(* IEC 61131-3 sources: mect_apps/TPAC1007_04_AA/Octopus_Head_PLC, 25 files *)

(* ---- Crosstable.gvl ---- *)
VAR_GLOBAL
PRODUCT_ID AT %QD0.4:UDINT;
SERIAL_NUMBER AT %QD0.8:UDINT;
TEST_ID AT %QW0.12:UINT;
TEST_STEP AT %QW0.16:UINT;
TEST_STEP_MAX AT %QW0.20:UINT;
TEST_DATE AT %QD0.24:UDINT;
TEST_TIME AT %QD0.28:UDINT;
TEST_DURATION AT %QD0.32:UDINT;
AUTOMATIC AT %IX0.772.0:BOOL;
DO_REPEAT AT %IX0.776.0:BOOL;
DO_RELOAD AT %IX0.780.0:BOOL;
STATUS AT %QW0.784:UINT;
RESULT AT %QW0.788:INT;
RESULTS_OK AT %QW0.792:UINT;
RESULTS_NG AT %QW0.796:UINT;
RTU_HeartBeat AT %ID0.832:UDINT;
RTU_DigOut_1 AT %QX0.840.0:BOOL;
RTU_DigOut_2 AT %QX0.844.0:BOOL;
RTU_DigOut_3 AT %QX0.848.0:BOOL;
RTU_DigOut_4 AT %QX0.852.0:BOOL;
RTU_DigOut_5 AT %QX0.856.0:BOOL;
RTU_DigOut_6 AT %QX0.860.0:BOOL;
RTU_DigOut_7 AT %QX0.864.0:BOOL;
RTU_DigOut_8 AT %QX0.868.0:BOOL;
RTU_DigOut_9 AT %QX0.872.0:BOOL;
RTU_DigOut_10 AT %QX0.876.0:BOOL;
RTU_DigOut_11 AT %QX0.880.0:BOOL;
RTU_DigOut_12 AT %QX0.884.0:BOOL;
RTU_DigOut_13 AT %QX0.888.0:BOOL;
RTU_DigOut_14 AT %QX0.892.0:BOOL;
RTU_DigOut_15 AT %QX0.896.0:BOOL;
RTU_DigOut_16 AT %QX0.900.0:BOOL;
RTU_DigIn_1 AT %IX0.908.0:BOOL;
RTU_DigIn_2 AT %IX0.912.0:BOOL;
RTU_DigIn_3 AT %IX0.916.0:BOOL;
RTU_DigIn_4 AT %IX0.920.0:BOOL;
RTU_DigIn_5 AT %IX0.924.0:BOOL;
RTU_DigIn_6 AT %IX0.928.0:BOOL;
RTU_DigIn_7 AT %IX0.932.0:BOOL;
RTU_DigIn_8 AT %IX0.936.0:BOOL;
RTU_DigIn_9 AT %IX0.940.0:BOOL;
RTU_DigIn_10 AT %IX0.944.0:BOOL;
RTU_DigIn_11 AT %IX0.948.0:BOOL;
RTU_DigIn_12 AT %IX0.952.0:BOOL;
RTU_DigIn_13 AT %IX0.956.0:BOOL;
RTU_DigIn_14 AT %IX0.960.0:BOOL;
RTU_DigIn_15 AT %IX0.964.0:BOOL;
RTU_DigIn_16 AT %IX0.968.0:BOOL;
RTU_Tamb AT %IW0.976:INT;
RTU_AnInConf_1 AT %QW0.980:UINT;
RTU_AnInConf_2 AT %QW0.984:UINT;
RTU_AnIn_1 AT %IW0.988:INT;
RTU_AnIn_2 AT %IW0.992:INT;
RTU_LocDigDir_1 AT %QX0.996.0:BOOL;
RTU_LocDigDir_2 AT %QX0.1000.0:BOOL;
RTU_LocDigDir_3 AT %QX0.1004.0:BOOL;
RTU_LocDigDir_4 AT %QX0.1008.0:BOOL;
RTU_LocDigDir_5 AT %QX0.1012.0:BOOL;
RTU_LocDigDir_6 AT %QX0.1016.0:BOOL;
RTU_LocDigDir_7 AT %QX0.1020.0:BOOL;
RTU_LocDigDir_8 AT %QX0.1024.0:BOOL;
RTU_LocDigIn_1 AT %IX0.1028.0:BOOL;
RTU_LocDigIn_2 AT %IX0.1032.0:BOOL;
RTU_LocDigIn_3 AT %IX0.1036.0:BOOL;
RTU_LocDigIn_4 AT %IX0.1040.0:BOOL;
RTU_LocDigIn_5 AT %IX0.1044.0:BOOL;
RTU_LocDigIn_6 AT %IX0.1048.0:BOOL;
RTU_LocDigIn_7 AT %IX0.1052.0:BOOL;
RTU_LocDigIn_8 AT %IX0.1056.0:BOOL;
RTU_LocDigOut_1 AT %QX0.1060.0:BOOL;
RTU_LocDigOut_2 AT %QX0.1064.0:BOOL;
RTU_LocDigOut_3 AT %QX0.1068.0:BOOL;
RTU_LocDigOut_4 AT %QX0.1072.0:BOOL;
RTU_LocDigOut_5 AT %QX0.1076.0:BOOL;
RTU_LocDigOut_6 AT %QX0.1080.0:BOOL;
RTU_LocDigOut_7 AT %QX0.1084.0:BOOL;
RTU_LocDigOut_8 AT %QX0.1088.0:BOOL;
TST_DigIn_1 AT %QX0.4004.0:BOOL;
TST_DigIn_2 AT %QX0.4008.0:BOOL;
TST_DigIn_3 AT %QX0.4012.0:BOOL;
TST_DigIn_4 AT %QX0.4016.0:BOOL;
TST_DigIn_5 AT %QX0.4020.0:BOOL;
TST_DigIn_6 AT %QX0.4024.0:BOOL;
TST_DigIn_7 AT %QX0.4028.0:BOOL;
TST_DigIn_8 AT %QX0.4032.0:BOOL;
TST_DigIn_9 AT %QX0.4036.0:BOOL;
TST_DigIn_10 AT %QX0.4040.0:BOOL;
TST_DigIn_11 AT %QX0.4044.0:BOOL;
TST_DigIn_12 AT %QX0.4048.0:BOOL;
TST_DigIn_13 AT %QX0.4052.0:BOOL;
TST_DigIn_14 AT %QX0.4056.0:BOOL;
TST_DigIn_15 AT %QX0.4060.0:BOOL;
TST_DigIn_16 AT %QX0.4064.0:BOOL;
VAL_DigIn_1 AT %QX0.4068.0:BOOL;
VAL_DigIn_2 AT %QX0.4072.0:BOOL;
VAL_DigIn_3 AT %QX0.4076.0:BOOL;
VAL_DigIn_4 AT %QX0.4080.0:BOOL;
VAL_DigIn_5 AT %QX0.4084.0:BOOL;
VAL_DigIn_6 AT %QX0.4088.0:BOOL;
VAL_DigIn_7 AT %QX0.4092.0:BOOL;
VAL_DigIn_8 AT %QX0.4096.0:BOOL;
VAL_DigIn_9 AT %QX0.4100.0:BOOL;
VAL_DigIn_10 AT %QX0.4104.0:BOOL;
VAL_DigIn_11 AT %QX0.4108.0:BOOL;
VAL_DigIn_12 AT %QX0.4112.0:BOOL;
VAL_DigIn_13 AT %QX0.4116.0:BOOL;
VAL_DigIn_14 AT %QX0.4120.0:BOOL;
VAL_DigIn_15 AT %QX0.4124.0:BOOL;
VAL_DigIn_16 AT %QX0.4128.0:BOOL;
RES_DigIn_1 AT %QX0.4132.0:BOOL;
RES_DigIn_2 AT %QX0.4136.0:BOOL;
RES_DigIn_3 AT %QX0.4140.0:BOOL;
RES_DigIn_4 AT %QX0.4144.0:BOOL;
RES_DigIn_5 AT %QX0.4148.0:BOOL;
RES_DigIn_6 AT %QX0.4152.0:BOOL;
RES_DigIn_7 AT %QX0.4156.0:BOOL;
RES_DigIn_8 AT %QX0.4160.0:BOOL;
RES_DigIn_9 AT %QX0.4164.0:BOOL;
RES_DigIn_10 AT %QX0.4168.0:BOOL;
RES_DigIn_11 AT %QX0.4172.0:BOOL;
RES_DigIn_12 AT %QX0.4176.0:BOOL;
RES_DigIn_13 AT %QX0.4180.0:BOOL;
RES_DigIn_14 AT %QX0.4184.0:BOOL;
RES_DigIn_15 AT %QX0.4188.0:BOOL;
RES_DigIn_16 AT %QX0.4192.0:BOOL;
OK_DigIn_1 AT %QX0.4196.0:BOOL;
OK_DigIn_2 AT %QX0.4200.0:BOOL;
OK_DigIn_3 AT %QX0.4204.0:BOOL;
OK_DigIn_4 AT %QX0.4208.0:BOOL;
OK_DigIn_5 AT %QX0.4212.0:BOOL;
OK_DigIn_6 AT %QX0.4216.0:BOOL;
OK_DigIn_7 AT %QX0.4220.0:BOOL;
OK_DigIn_8 AT %QX0.4224.0:BOOL;
OK_DigIn_9 AT %QX0.4228.0:BOOL;
OK_DigIn_10 AT %QX0.4232.0:BOOL;
OK_DigIn_11 AT %QX0.4236.0:BOOL;
OK_DigIn_12 AT %QX0.4240.0:BOOL;
OK_DigIn_13 AT %QX0.4244.0:BOOL;
OK_DigIn_14 AT %QX0.4248.0:BOOL;
OK_DigIn_15 AT %QX0.4252.0:BOOL;
OK_DigIn_16 AT %QX0.4256.0:BOOL;
TST_DigOut_1 AT %QX0.4260.0:BOOL;
TST_DigOut_2 AT %QX0.4264.0:BOOL;
TST_DigOut_3 AT %QX0.4268.0:BOOL;
TST_DigOut_4 AT %QX0.4272.0:BOOL;
TST_DigOut_5 AT %QX0.4276.0:BOOL;
TST_DigOut_6 AT %QX0.4280.0:BOOL;
TST_DigOut_7 AT %QX0.4284.0:BOOL;
TST_DigOut_8 AT %QX0.4288.0:BOOL;
TST_DigOut_9 AT %QX0.4292.0:BOOL;
TST_DigOut_10 AT %QX0.4296.0:BOOL;
TST_DigOut_11 AT %QX0.4300.0:BOOL;
TST_DigOut_12 AT %QX0.4304.0:BOOL;
TST_DigOut_13 AT %QX0.4308.0:BOOL;
TST_DigOut_14 AT %QX0.4312.0:BOOL;
TST_DigOut_15 AT %QX0.4316.0:BOOL;
TST_DigOut_16 AT %QX0.4320.0:BOOL;
VAL_DigOut_1 AT %QX0.4324.0:BOOL;
VAL_DigOut_2 AT %QX0.4328.0:BOOL;
VAL_DigOut_3 AT %QX0.4332.0:BOOL;
VAL_DigOut_4 AT %QX0.4336.0:BOOL;
VAL_DigOut_5 AT %QX0.4340.0:BOOL;
VAL_DigOut_6 AT %QX0.4344.0:BOOL;
VAL_DigOut_7 AT %QX0.4348.0:BOOL;
VAL_DigOut_8 AT %QX0.4352.0:BOOL;
VAL_DigOut_9 AT %QX0.4356.0:BOOL;
VAL_DigOut_10 AT %QX0.4360.0:BOOL;
VAL_DigOut_11 AT %QX0.4364.0:BOOL;
VAL_DigOut_12 AT %QX0.4368.0:BOOL;
VAL_DigOut_13 AT %QX0.4372.0:BOOL;
VAL_DigOut_14 AT %QX0.4376.0:BOOL;
VAL_DigOut_15 AT %QX0.4380.0:BOOL;
VAL_DigOut_16 AT %QX0.4384.0:BOOL;
RES_DigOut_1 AT %QX0.4388.0:BOOL;
RES_DigOut_2 AT %QX0.4392.0:BOOL;
RES_DigOut_3 AT %QX0.4396.0:BOOL;
RES_DigOut_4 AT %QX0.4400.0:BOOL;
RES_DigOut_5 AT %QX0.4404.0:BOOL;
RES_DigOut_6 AT %QX0.4408.0:BOOL;
RES_DigOut_7 AT %QX0.4412.0:BOOL;
RES_DigOut_8 AT %QX0.4416.0:BOOL;
RES_DigOut_9 AT %QX0.4420.0:BOOL;
RES_DigOut_10 AT %QX0.4424.0:BOOL;
RES_DigOut_11 AT %QX0.4428.0:BOOL;
RES_DigOut_12 AT %QX0.4432.0:BOOL;
RES_DigOut_13 AT %QX0.4436.0:BOOL;
RES_DigOut_14 AT %QX0.4440.0:BOOL;
RES_DigOut_15 AT %QX0.4444.0:BOOL;
RES_DigOut_16 AT %QX0.4448.0:BOOL;
OK_DigOut_1 AT %QX0.4452.0:BOOL;
OK_DigOut_2 AT %QX0.4456.0:BOOL;
OK_DigOut_3 AT %QX0.4460.0:BOOL;
OK_DigOut_4 AT %QX0.4464.0:BOOL;
OK_DigOut_5 AT %QX0.4468.0:BOOL;
OK_DigOut_6 AT %QX0.4472.0:BOOL;
OK_DigOut_7 AT %QX0.4476.0:BOOL;
OK_DigOut_8 AT %QX0.4480.0:BOOL;
OK_DigOut_9 AT %QX0.4484.0:BOOL;
OK_DigOut_10 AT %QX0.4488.0:BOOL;
OK_DigOut_11 AT %QX0.4492.0:BOOL;
OK_DigOut_12 AT %QX0.4496.0:BOOL;
OK_DigOut_13 AT %QX0.4500.0:BOOL;
OK_DigOut_14 AT %QX0.4504.0:BOOL;
OK_DigOut_15 AT %QX0.4508.0:BOOL;
OK_DigOut_16 AT %QX0.4512.0:BOOL;
TST_AnIn_1 AT %QX0.4516.0:BOOL;
TST_AnIn_2 AT %QX0.4520.0:BOOL;
TST_AnIn_3 AT %QX0.4524.0:BOOL;
TST_AnIn_4 AT %QX0.4528.0:BOOL;
TST_AnIn_5 AT %QX0.4532.0:BOOL;
TST_AnIn_6 AT %QX0.4536.0:BOOL;
TST_AnIn_7 AT %QX0.4540.0:BOOL;
TST_AnIn_8 AT %QX0.4544.0:BOOL;
TST_AnIn_9 AT %QX0.4548.0:BOOL;
TST_AnIn_10 AT %QX0.4552.0:BOOL;
TST_AnIn_11 AT %QX0.4556.0:BOOL;
TST_AnIn_12 AT %QX0.4560.0:BOOL;
VAL_AnIn_1 AT %QW0.4564:INT;
VAL_AnIn_2 AT %QW0.4568:INT;
VAL_AnIn_3 AT %QW0.4572:INT;
VAL_AnIn_4 AT %QW0.4576:INT;
VAL_AnIn_5 AT %QW0.4580:INT;
VAL_AnIn_6 AT %QW0.4584:INT;
VAL_AnIn_7 AT %QW0.4588:INT;
VAL_AnIn_8 AT %QW0.4592:INT;
VAL_AnIn_9 AT %QW0.4596:INT;
VAL_AnIn_10 AT %QW0.4600:INT;
VAL_AnIn_11 AT %QW0.4604:INT;
VAL_AnIn_12 AT %QW0.4608:INT;
VAL_AnInConf_1 AT %QW0.4612:UINT;
VAL_AnInConf_2 AT %QW0.4616:UINT;
VAL_AnInConf_3 AT %QW0.4620:UINT;
VAL_AnInConf_4 AT %QW0.4624:UINT;
VAL_AnInConf_5 AT %QW0.4628:UINT;
VAL_AnInConf_6 AT %QW0.4632:UINT;
VAL_AnInConf_7 AT %QW0.4636:UINT;
VAL_AnInConf_8 AT %QW0.4640:UINT;
VAL_AnInConf_9 AT %QW0.4644:UINT;
VAL_AnInConf_10 AT %QW0.4648:UINT;
VAL_AnInConf_11 AT %QW0.4652:UINT;
VAL_AnInConf_12 AT %QW0.4656:UINT;
VAL_AnInFltr_1 AT %QW0.4660:UINT;
VAL_AnInFltr_2 AT %QW0.4664:UINT;
VAL_AnInFltr_3 AT %QW0.4668:UINT;
VAL_AnInFltr_4 AT %QW0.4672:UINT;
VAL_AnInFltr_5 AT %QW0.4676:UINT;
VAL_AnInFltr_6 AT %QW0.4680:UINT;
VAL_AnInFltr_7 AT %QW0.4684:UINT;
VAL_AnInFltr_8 AT %QW0.4688:UINT;
VAL_AnInFltr_9 AT %QW0.4692:UINT;
VAL_AnInFltr_10 AT %QW0.4696:UINT;
VAL_AnInFltr_11 AT %QW0.4700:UINT;
VAL_AnInFltr_12 AT %QW0.4704:UINT;
RES_AnIn_1 AT %QW0.4708:INT;
RES_AnIn_2 AT %QW0.4712:INT;
RES_AnIn_3 AT %QW0.4716:INT;
RES_AnIn_4 AT %QW0.4720:INT;
RES_AnIn_5 AT %QW0.4724:INT;
RES_AnIn_6 AT %QW0.4728:INT;
RES_AnIn_7 AT %QW0.4732:INT;
RES_AnIn_8 AT %QW0.4736:INT;
RES_AnIn_9 AT %QW0.4740:INT;
RES_AnIn_10 AT %QW0.4744:INT;
RES_AnIn_11 AT %QW0.4748:INT;
RES_AnIn_12 AT %QW0.4752:INT;
RES_AnInStts_1 AT %QW0.4756:INT;
RES_AnInStts_2 AT %QW0.4760:INT;
RES_AnInStts_3 AT %QW0.4764:INT;
RES_AnInStts_4 AT %QW0.4768:INT;
RES_AnInStts_5 AT %QW0.4772:INT;
RES_AnInStts_6 AT %QW0.4776:INT;
RES_AnInStts_7 AT %QW0.4780:INT;
RES_AnInStts_8 AT %QW0.4784:INT;
RES_AnInStts_9 AT %QW0.4788:INT;
RES_AnInStts_10 AT %QW0.4792:INT;
RES_AnInStts_11 AT %QW0.4796:INT;
RES_AnInStts_12 AT %QW0.4800:INT;
OK_AnIn_1 AT %QX0.4804.0:BOOL;
OK_AnIn_2 AT %QX0.4808.0:BOOL;
OK_AnIn_3 AT %QX0.4812.0:BOOL;
OK_AnIn_4 AT %QX0.4816.0:BOOL;
OK_AnIn_5 AT %QX0.4820.0:BOOL;
OK_AnIn_6 AT %QX0.4824.0:BOOL;
OK_AnIn_7 AT %QX0.4828.0:BOOL;
OK_AnIn_8 AT %QX0.4832.0:BOOL;
OK_AnIn_9 AT %QX0.4836.0:BOOL;
OK_AnIn_10 AT %QX0.4840.0:BOOL;
OK_AnIn_11 AT %QX0.4844.0:BOOL;
OK_AnIn_12 AT %QX0.4848.0:BOOL;
TST_AnOut_1 AT %QX0.4852.0:BOOL;
TST_AnOut_2 AT %QX0.4856.0:BOOL;
TST_AnOut_3 AT %QX0.4860.0:BOOL;
TST_AnOut_4 AT %QX0.4864.0:BOOL;
VAL_AnOut_1 AT %QW0.4868:INT;
VAL_AnOut_2 AT %QW0.4872:INT;
VAL_AnOut_3 AT %QW0.4876:INT;
VAL_AnOut_4 AT %QW0.4880:INT;
VAL_AnOutConf_1 AT %QW0.4884:UINT;
VAL_AnOutConf_2 AT %QW0.4888:UINT;
VAL_AnOutConf_3 AT %QW0.4892:UINT;
VAL_AnOutConf_4 AT %QW0.4896:UINT;
RES_AnOut_1 AT %QW0.4900:INT;
RES_AnOut_2 AT %QW0.4904:INT;
RES_AnOut_3 AT %QW0.4908:INT;
RES_AnOut_4 AT %QW0.4912:INT;
RES_AnOutStts_1 AT %QW0.4916:INT;
RES_AnOutStts_2 AT %QW0.4920:INT;
RES_AnOutStts_3 AT %QW0.4924:INT;
RES_AnOutStts_4 AT %QW0.4928:INT;
OK_AnOut_1 AT %QX0.4932.0:BOOL;
OK_AnOut_2 AT %QX0.4936.0:BOOL;
OK_AnOut_3 AT %QX0.4940.0:BOOL;
OK_AnOut_4 AT %QX0.4944.0:BOOL;
TST_Tamb AT %QX0.4948.0:BOOL;
TST_RPM AT %QX0.4952.0:BOOL;
TST_VCC_set AT %QX0.4956.0:BOOL;
TST_mA_max AT %QX0.4960.0:BOOL;
TST_VCC_fbk AT %QX0.4964.0:BOOL;
TST_mA_fbk AT %QX0.4968.0:BOOL;
TST_FWrevision AT %QX0.4972.0:BOOL;
TST_HWconfig AT %QX0.4976.0:BOOL;
VAL_Tamb AT %QW0.4980:INT;
VAL_RPM AT %QW0.4984:UINT;
VAL_VCC_set AT %QW0.4988:INT;
VAL_mA_max AT %QW0.4992:INT;
VAL_VCC_fbk AT %QW0.4996:INT;
VAL_mA_fbk AT %QW0.5000:INT;
VAL_FWrevision AT %QW0.5004:UINT;
VAL_HWconfig AT %QW0.5008:UINT;
RES_Tamb AT %QW0.5012:INT;
RES_RPM AT %QW0.5016:UINT;
RES_VCC_set AT %QW0.5020:INT;
RES_mA_max AT %QW0.5024:INT;
RES_VCC_fbk AT %QW0.5028:INT;
RES_mA_fbk AT %QW0.5032:INT;
RES_FWrevision AT %QW0.5036:UINT;
RES_HWconfig AT %QW0.5040:UINT;
OK_Tamb AT %QX0.5044.0:BOOL;
OK_RPM AT %QX0.5048.0:BOOL;
OK_VCC_set AT %QX0.5052.0:BOOL;
OK_mA_max AT %QX0.5056.0:BOOL;
OK_VCC_fbk AT %QX0.5060.0:BOOL;
OK_mA_fbk AT %QX0.5064.0:BOOL;
OK_FWrevision AT %QX0.5068.0:BOOL;
OK_HWconfig AT %QX0.5072.0:BOOL;
TST_RTUS_WR AT %QX0.5076.0:BOOL;
TST_RTUS_RD AT %QX0.5080.0:BOOL;
TST_RTU1_WR AT %QX0.5084.0:BOOL;
TST_RTU1_RD AT %QX0.5088.0:BOOL;
TST_RTU3_WR AT %QX0.5092.0:BOOL;
TST_RTU3_RD AT %QX0.5096.0:BOOL;
TST_CAN1_WR AT %QX0.5100.0:BOOL;
TST_CAN1_RD AT %QX0.5104.0:BOOL;
VAL_RTUS_WR AT %QX0.5108.0:BOOL;
VAL_RTUS_RD AT %QX0.5112.0:BOOL;
VAL_RTU1_WR AT %QX0.5116.0:BOOL;
VAL_RTU1_RD AT %QX0.5120.0:BOOL;
VAL_RTU3_WR AT %QX0.5124.0:BOOL;
VAL_RTU3_RD AT %QX0.5128.0:BOOL;
VAL_CAN1_WR AT %QX0.5132.0:BOOL;
VAL_CAN1_RD AT %QX0.5136.0:BOOL;
RES_RTUS_WR AT %QX0.5140.0:BOOL;
RES_RTUS_RD AT %QX0.5144.0:BOOL;
RES_RTU1_WR AT %QX0.5148.0:BOOL;
RES_RTU1_RD AT %QX0.5152.0:BOOL;
RES_RTU3_WR AT %QX0.5156.0:BOOL;
RES_RTU3_RD AT %QX0.5160.0:BOOL;
RES_CAN1_WR AT %QX0.5164.0:BOOL;
RES_CAN1_RD AT %QX0.5168.0:BOOL;
OK_RTUS_WR AT %QX0.5172.0:BOOL;
OK_RTUS_RD AT %QX0.5176.0:BOOL;
OK_RTU1_WR AT %QX0.5180.0:BOOL;
OK_RTU1_RD AT %QX0.5184.0:BOOL;
OK_RTU3_WR AT %QX0.5188.0:BOOL;
OK_RTU3_RD AT %QX0.5192.0:BOOL;
OK_CAN1_WR AT %QX0.5196.0:BOOL;
OK_CAN1_RD AT %QX0.5200.0:BOOL;
TEST2_COMMAND AT %QW0.12000:UINT;
TST2_DigIn_1 AT %QX0.12004.0:BOOL;
TST2_DigIn_2 AT %QX0.12008.0:BOOL;
TST2_DigIn_3 AT %QX0.12012.0:BOOL;
TST2_DigIn_4 AT %QX0.12016.0:BOOL;
TST2_DigIn_5 AT %QX0.12020.0:BOOL;
TST2_DigIn_6 AT %QX0.12024.0:BOOL;
TST2_DigIn_7 AT %QX0.12028.0:BOOL;
TST2_DigIn_8 AT %QX0.12032.0:BOOL;
TST2_DigIn_9 AT %QX0.12036.0:BOOL;
TST2_DigIn_10 AT %QX0.12040.0:BOOL;
TST2_DigIn_11 AT %QX0.12044.0:BOOL;
TST2_DigIn_12 AT %QX0.12048.0:BOOL;
TST2_DigIn_13 AT %QX0.12052.0:BOOL;
TST2_DigIn_14 AT %QX0.12056.0:BOOL;
TST2_DigIn_15 AT %QX0.12060.0:BOOL;
TST2_DigIn_16 AT %QX0.12064.0:BOOL;
VAL2_DigIn_1 AT %QX0.12068.0:BOOL;
VAL2_DigIn_2 AT %QX0.12072.0:BOOL;
VAL2_DigIn_3 AT %QX0.12076.0:BOOL;
VAL2_DigIn_4 AT %QX0.12080.0:BOOL;
VAL2_DigIn_5 AT %QX0.12084.0:BOOL;
VAL2_DigIn_6 AT %QX0.12088.0:BOOL;
VAL2_DigIn_7 AT %QX0.12092.0:BOOL;
VAL2_DigIn_8 AT %QX0.12096.0:BOOL;
VAL2_DigIn_9 AT %QX0.12100.0:BOOL;
VAL2_DigIn_10 AT %QX0.12104.0:BOOL;
VAL2_DigIn_11 AT %QX0.12108.0:BOOL;
VAL2_DigIn_12 AT %QX0.12112.0:BOOL;
VAL2_DigIn_13 AT %QX0.12116.0:BOOL;
VAL2_DigIn_14 AT %QX0.12120.0:BOOL;
VAL2_DigIn_15 AT %QX0.12124.0:BOOL;
VAL2_DigIn_16 AT %QX0.12128.0:BOOL;
RES2_DigIn_1 AT %IX0.12132.0:BOOL;
RES2_DigIn_2 AT %IX0.12136.0:BOOL;
RES2_DigIn_3 AT %IX0.12140.0:BOOL;
RES2_DigIn_4 AT %IX0.12144.0:BOOL;
RES2_DigIn_5 AT %IX0.12148.0:BOOL;
RES2_DigIn_6 AT %IX0.12152.0:BOOL;
RES2_DigIn_7 AT %IX0.12156.0:BOOL;
RES2_DigIn_8 AT %IX0.12160.0:BOOL;
RES2_DigIn_9 AT %IX0.12164.0:BOOL;
RES2_DigIn_10 AT %IX0.12168.0:BOOL;
RES2_DigIn_11 AT %IX0.12172.0:BOOL;
RES2_DigIn_12 AT %IX0.12176.0:BOOL;
RES2_DigIn_13 AT %IX0.12180.0:BOOL;
RES2_DigIn_14 AT %IX0.12184.0:BOOL;
RES2_DigIn_15 AT %IX0.12188.0:BOOL;
RES2_DigIn_16 AT %IX0.12192.0:BOOL;
TST2_DigOut_1 AT %QX0.12196.0:BOOL;
TST2_DigOut_2 AT %QX0.12200.0:BOOL;
TST2_DigOut_3 AT %QX0.12204.0:BOOL;
TST2_DigOut_4 AT %QX0.12208.0:BOOL;
TST2_DigOut_5 AT %QX0.12212.0:BOOL;
TST2_DigOut_6 AT %QX0.12216.0:BOOL;
TST2_DigOut_7 AT %QX0.12220.0:BOOL;
TST2_DigOut_8 AT %QX0.12224.0:BOOL;
TST2_DigOut_9 AT %QX0.12228.0:BOOL;
TST2_DigOut_10 AT %QX0.12232.0:BOOL;
TST2_DigOut_11 AT %QX0.12236.0:BOOL;
TST2_DigOut_12 AT %QX0.12240.0:BOOL;
TST2_DigOut_13 AT %QX0.12244.0:BOOL;
TST2_DigOut_14 AT %QX0.12248.0:BOOL;
TST2_DigOut_15 AT %QX0.12252.0:BOOL;
TST2_DigOut_16 AT %QX0.12256.0:BOOL;
VAL2_DigOut_1 AT %QX0.12260.0:BOOL;
VAL2_DigOut_2 AT %QX0.12264.0:BOOL;
VAL2_DigOut_3 AT %QX0.12268.0:BOOL;
VAL2_DigOut_4 AT %QX0.12272.0:BOOL;
VAL2_DigOut_5 AT %QX0.12276.0:BOOL;
VAL2_DigOut_6 AT %QX0.12280.0:BOOL;
VAL2_DigOut_7 AT %QX0.12284.0:BOOL;
VAL2_DigOut_8 AT %QX0.12288.0:BOOL;
VAL2_DigOut_9 AT %QX0.12292.0:BOOL;
VAL2_DigOut_10 AT %QX0.12296.0:BOOL;
VAL2_DigOut_11 AT %QX0.12300.0:BOOL;
VAL2_DigOut_12 AT %QX0.12304.0:BOOL;
VAL2_DigOut_13 AT %QX0.12308.0:BOOL;
VAL2_DigOut_14 AT %QX0.12312.0:BOOL;
VAL2_DigOut_15 AT %QX0.12316.0:BOOL;
VAL2_DigOut_16 AT %QX0.12320.0:BOOL;
TST2_AnIn_1 AT %QX0.12324.0:BOOL;
TST2_AnIn_2 AT %QX0.12328.0:BOOL;
TST2_AnIn_3 AT %QX0.12332.0:BOOL;
TST2_AnIn_4 AT %QX0.12336.0:BOOL;
TST2_AnIn_5 AT %QX0.12340.0:BOOL;
TST2_AnIn_6 AT %QX0.12344.0:BOOL;
TST2_AnIn_7 AT %QX0.12348.0:BOOL;
TST2_AnIn_8 AT %QX0.12352.0:BOOL;
TST2_AnIn_9 AT %QX0.12356.0:BOOL;
TST2_AnIn_10 AT %QX0.12360.0:BOOL;
TST2_AnIn_11 AT %QX0.12364.0:BOOL;
TST2_AnIn_12 AT %QX0.12368.0:BOOL;
VAL2_AnIn_1 AT %QW0.12372:INT;
VAL2_AnIn_2 AT %QW0.12376:INT;
VAL2_AnIn_3 AT %QW0.12380:INT;
VAL2_AnIn_4 AT %QW0.12384:INT;
VAL2_AnIn_5 AT %QW0.12388:INT;
VAL2_AnIn_6 AT %QW0.12392:INT;
VAL2_AnIn_7 AT %QW0.12396:INT;
VAL2_AnIn_8 AT %QW0.12400:INT;
VAL2_AnIn_9 AT %QW0.12404:INT;
VAL2_AnIn_10 AT %QW0.12408:INT;
VAL2_AnIn_11 AT %QW0.12412:INT;
VAL2_AnIn_12 AT %QW0.12416:INT;
VAL2_AnInConf_1 AT %QW0.12420:UINT;
VAL2_AnInConf_2 AT %QW0.12424:UINT;
VAL2_AnInConf_3 AT %QW0.12428:UINT;
VAL2_AnInConf_4 AT %QW0.12432:UINT;
VAL2_AnInConf_5 AT %QW0.12436:UINT;
VAL2_AnInConf_6 AT %QW0.12440:UINT;
VAL2_AnInConf_7 AT %QW0.12444:UINT;
VAL2_AnInConf_8 AT %QW0.12448:UINT;
VAL2_AnInConf_9 AT %QW0.12452:UINT;
VAL2_AnInConf_10 AT %QW0.12456:UINT;
VAL2_AnInConf_11 AT %QW0.12460:UINT;
VAL2_AnInConf_12 AT %QW0.12464:UINT;
VAL2_AnInFltr_1 AT %QW0.12468:UINT;
VAL2_AnInFltr_2 AT %QW0.12472:UINT;
VAL2_AnInFltr_3 AT %QW0.12476:UINT;
VAL2_AnInFltr_4 AT %QW0.12480:UINT;
VAL2_AnInFltr_5 AT %QW0.12484:UINT;
VAL2_AnInFltr_6 AT %QW0.12488:UINT;
VAL2_AnInFltr_7 AT %QW0.12492:UINT;
VAL2_AnInFltr_8 AT %QW0.12496:UINT;
VAL2_AnInFltr_9 AT %QW0.12500:UINT;
VAL2_AnInFltr_10 AT %QW0.12504:UINT;
VAL2_AnInFltr_11 AT %QW0.12508:UINT;
VAL2_AnInFltr_12 AT %QW0.12512:UINT;
RES2_AnIn_1 AT %IW0.12516:INT;
RES2_AnIn_2 AT %IW0.12520:INT;
RES2_AnIn_3 AT %IW0.12524:INT;
RES2_AnIn_4 AT %IW0.12528:INT;
RES2_AnIn_5 AT %IW0.12532:INT;
RES2_AnIn_6 AT %IW0.12536:INT;
RES2_AnIn_7 AT %IW0.12540:INT;
RES2_AnIn_8 AT %IW0.12544:INT;
RES2_AnIn_9 AT %IW0.12548:INT;
RES2_AnIn_10 AT %IW0.12552:INT;
RES2_AnIn_11 AT %IW0.12556:INT;
RES2_AnIn_12 AT %IW0.12560:INT;
RES2_AnInStts_1 AT %IW0.12564:INT;
RES2_AnInStts_2 AT %IW0.12568:INT;
RES2_AnInStts_3 AT %IW0.12572:INT;
RES2_AnInStts_4 AT %IW0.12576:INT;
RES2_AnInStts_5 AT %IW0.12580:INT;
RES2_AnInStts_6 AT %IW0.12584:INT;
RES2_AnInStts_7 AT %IW0.12588:INT;
RES2_AnInStts_8 AT %IW0.12592:INT;
RES2_AnInStts_9 AT %IW0.12596:INT;
RES2_AnInStts_10 AT %IW0.12600:INT;
RES2_AnInStts_11 AT %IW0.12604:INT;
RES2_AnInStts_12 AT %IW0.12608:INT;
TST2_AnOut_1 AT %QX0.12612.0:BOOL;
TST2_AnOut_2 AT %QX0.12616.0:BOOL;
TST2_AnOut_3 AT %QX0.12620.0:BOOL;
TST2_AnOut_4 AT %QX0.12624.0:BOOL;
VAL2_AnOut_1 AT %QW0.12628:INT;
VAL2_AnOut_2 AT %QW0.12632:INT;
VAL2_AnOut_3 AT %QW0.12636:INT;
VAL2_AnOut_4 AT %QW0.12640:INT;
VAL2_AnOutConf_1 AT %QW0.12644:UINT;
VAL2_AnOutConf_2 AT %QW0.12648:UINT;
VAL2_AnOutConf_3 AT %QW0.12652:UINT;
VAL2_AnOutConf_4 AT %QW0.12656:UINT;
RES2_AnOutStts_1 AT %IW0.12660:INT;
RES2_AnOutStts_2 AT %IW0.12664:INT;
RES2_AnOutStts_3 AT %IW0.12668:INT;
RES2_AnOutStts_4 AT %IW0.12672:INT;
TST2_Tamb AT %QX0.12676.0:BOOL;
TST2_RPM AT %QX0.12680.0:BOOL;
TST2_FWrevision AT %QX0.12684.0:BOOL;
TST2_HWconfig AT %QX0.12688.0:BOOL;
VAL2_Tamb AT %QW0.12692:INT;
VAL2_RPM AT %QW0.12696:UINT;
VAL2_FWrevision AT %QW0.12700:UINT;
VAL2_HWconfig AT %QW0.12704:UINT;
RES2_Tamb AT %IW0.12708:INT;
RES2_RPM AT %IW0.12712:UINT;
RES2_FWrevision AT %IW0.12716:UINT;
RES2_HWconfig AT %IW0.12720:UINT;
TST2_RTUS_WR AT %QX0.12724.0:BOOL;
TST2_RTUS_RD AT %QX0.12728.0:BOOL;
TST2_RTU1_WR AT %QX0.12732.0:BOOL;
TST2_RTU1_RD AT %QX0.12736.0:BOOL;
TST2_RTU3_WR AT %QX0.12740.0:BOOL;
TST2_RTU3_RD AT %QX0.12744.0:BOOL;
TST2_CAN1_WR AT %QX0.12748.0:BOOL;
TST2_CAN1_RD AT %QX0.12752.0:BOOL;
VAL2_RTUS_WR AT %QX0.12756.0:BOOL;
VAL2_RTUS_RD AT %QX0.12760.0:BOOL;
VAL2_RTU1_WR AT %QX0.12764.0:BOOL;
VAL2_RTU1_RD AT %QX0.12768.0:BOOL;
VAL2_RTU3_WR AT %QX0.12772.0:BOOL;
VAL2_RTU3_RD AT %QX0.12776.0:BOOL;
VAL2_CAN1_WR AT %QX0.12780.0:BOOL;
VAL2_CAN1_RD AT %QX0.12784.0:BOOL;
RES2_RTUS_WR AT %QX0.12788.0:BOOL;
RES2_RTUS_RD AT %QX0.12792.0:BOOL;
RES2_RTU1_WR AT %QX0.12796.0:BOOL;
RES2_RTU1_RD AT %QX0.12800.0:BOOL;
RES2_RTU3_WR AT %QX0.12804.0:BOOL;
RES2_RTU3_RD AT %QX0.12808.0:BOOL;
RES2_CAN1_WR AT %QX0.12812.0:BOOL;
RES2_CAN1_RD AT %QX0.12816.0:BOOL;
TEST2_STATUS AT %IW0.12820:UINT;
TESTx_COMMAND AT %QW0.16000:UINT;
TSTx_DigIn_1 AT %QX0.16004.0:BOOL;
TSTx_DigIn_2 AT %QX0.16008.0:BOOL;
TSTx_DigIn_3 AT %QX0.16012.0:BOOL;
TSTx_DigIn_4 AT %QX0.16016.0:BOOL;
TSTx_DigIn_5 AT %QX0.16020.0:BOOL;
TSTx_DigIn_6 AT %QX0.16024.0:BOOL;
TSTx_DigIn_7 AT %QX0.16028.0:BOOL;
TSTx_DigIn_8 AT %QX0.16032.0:BOOL;
TSTx_DigIn_9 AT %QX0.16036.0:BOOL;
TSTx_DigIn_10 AT %QX0.16040.0:BOOL;
TSTx_DigIn_11 AT %QX0.16044.0:BOOL;
TSTx_DigIn_12 AT %QX0.16048.0:BOOL;
TSTx_DigIn_13 AT %QX0.16052.0:BOOL;
TSTx_DigIn_14 AT %QX0.16056.0:BOOL;
TSTx_DigIn_15 AT %QX0.16060.0:BOOL;
TSTx_DigIn_16 AT %QX0.16064.0:BOOL;
VALx_DigIn_1 AT %QX0.16068.0:BOOL;
VALx_DigIn_2 AT %QX0.16072.0:BOOL;
VALx_DigIn_3 AT %QX0.16076.0:BOOL;
VALx_DigIn_4 AT %QX0.16080.0:BOOL;
VALx_DigIn_5 AT %QX0.16084.0:BOOL;
VALx_DigIn_6 AT %QX0.16088.0:BOOL;
VALx_DigIn_7 AT %QX0.16092.0:BOOL;
VALx_DigIn_8 AT %QX0.16096.0:BOOL;
VALx_DigIn_9 AT %QX0.16100.0:BOOL;
VALx_DigIn_10 AT %QX0.16104.0:BOOL;
VALx_DigIn_11 AT %QX0.16108.0:BOOL;
VALx_DigIn_12 AT %QX0.16112.0:BOOL;
VALx_DigIn_13 AT %QX0.16116.0:BOOL;
VALx_DigIn_14 AT %QX0.16120.0:BOOL;
VALx_DigIn_15 AT %QX0.16124.0:BOOL;
VALx_DigIn_16 AT %QX0.16128.0:BOOL;
RESx_DigIn_1 AT %IX0.16132.0:BOOL;
RESx_DigIn_2 AT %IX0.16136.0:BOOL;
RESx_DigIn_3 AT %IX0.16140.0:BOOL;
RESx_DigIn_4 AT %IX0.16144.0:BOOL;
RESx_DigIn_5 AT %IX0.16148.0:BOOL;
RESx_DigIn_6 AT %IX0.16152.0:BOOL;
RESx_DigIn_7 AT %IX0.16156.0:BOOL;
RESx_DigIn_8 AT %IX0.16160.0:BOOL;
RESx_DigIn_9 AT %IX0.16164.0:BOOL;
RESx_DigIn_10 AT %IX0.16168.0:BOOL;
RESx_DigIn_11 AT %IX0.16172.0:BOOL;
RESx_DigIn_12 AT %IX0.16176.0:BOOL;
RESx_DigIn_13 AT %IX0.16180.0:BOOL;
RESx_DigIn_14 AT %IX0.16184.0:BOOL;
RESx_DigIn_15 AT %IX0.16188.0:BOOL;
RESx_DigIn_16 AT %IX0.16192.0:BOOL;
TSTx_DigOut_1 AT %QX0.16196.0:BOOL;
TSTx_DigOut_2 AT %QX0.16200.0:BOOL;
TSTx_DigOut_3 AT %QX0.16204.0:BOOL;
TSTx_DigOut_4 AT %QX0.16208.0:BOOL;
TSTx_DigOut_5 AT %QX0.16212.0:BOOL;
TSTx_DigOut_6 AT %QX0.16216.0:BOOL;
TSTx_DigOut_7 AT %QX0.16220.0:BOOL;
TSTx_DigOut_8 AT %QX0.16224.0:BOOL;
TSTx_DigOut_9 AT %QX0.16228.0:BOOL;
TSTx_DigOut_10 AT %QX0.16232.0:BOOL;
TSTx_DigOut_11 AT %QX0.16236.0:BOOL;
TSTx_DigOut_12 AT %QX0.16240.0:BOOL;
TSTx_DigOut_13 AT %QX0.16244.0:BOOL;
TSTx_DigOut_14 AT %QX0.16248.0:BOOL;
TSTx_DigOut_15 AT %QX0.16252.0:BOOL;
TSTx_DigOut_16 AT %QX0.16256.0:BOOL;
VALx_DigOut_1 AT %QX0.16260.0:BOOL;
VALx_DigOut_2 AT %QX0.16264.0:BOOL;
VALx_DigOut_3 AT %QX0.16268.0:BOOL;
VALx_DigOut_4 AT %QX0.16272.0:BOOL;
VALx_DigOut_5 AT %QX0.16276.0:BOOL;
VALx_DigOut_6 AT %QX0.16280.0:BOOL;
VALx_DigOut_7 AT %QX0.16284.0:BOOL;
VALx_DigOut_8 AT %QX0.16288.0:BOOL;
VALx_DigOut_9 AT %QX0.16292.0:BOOL;
VALx_DigOut_10 AT %QX0.16296.0:BOOL;
VALx_DigOut_11 AT %QX0.16300.0:BOOL;
VALx_DigOut_12 AT %QX0.16304.0:BOOL;
VALx_DigOut_13 AT %QX0.16308.0:BOOL;
VALx_DigOut_14 AT %QX0.16312.0:BOOL;
VALx_DigOut_15 AT %QX0.16316.0:BOOL;
VALx_DigOut_16 AT %QX0.16320.0:BOOL;
TSTx_AnIn_1 AT %QX0.16324.0:BOOL;
TSTx_AnIn_2 AT %QX0.16328.0:BOOL;
TSTx_AnIn_3 AT %QX0.16332.0:BOOL;
TSTx_AnIn_4 AT %QX0.16336.0:BOOL;
TSTx_AnIn_5 AT %QX0.16340.0:BOOL;
TSTx_AnIn_6 AT %QX0.16344.0:BOOL;
TSTx_AnIn_7 AT %QX0.16348.0:BOOL;
TSTx_AnIn_8 AT %QX0.16352.0:BOOL;
TSTx_AnIn_9 AT %QX0.16356.0:BOOL;
TSTx_AnIn_10 AT %QX0.16360.0:BOOL;
TSTx_AnIn_11 AT %QX0.16364.0:BOOL;
TSTx_AnIn_12 AT %QX0.16368.0:BOOL;
VALx_AnIn_1 AT %QW0.16372:INT;
VALx_AnIn_2 AT %QW0.16376:INT;
VALx_AnIn_3 AT %QW0.16380:INT;
VALx_AnIn_4 AT %QW0.16384:INT;
VALx_AnIn_5 AT %QW0.16388:INT;
VALx_AnIn_6 AT %QW0.16392:INT;
VALx_AnIn_7 AT %QW0.16396:INT;
VALx_AnIn_8 AT %QW0.16400:INT;
VALx_AnIn_9 AT %QW0.16404:INT;
VALx_AnIn_10 AT %QW0.16408:INT;
VALx_AnIn_11 AT %QW0.16412:INT;
VALx_AnIn_12 AT %QW0.16416:INT;
VALx_AnInConf_1 AT %QW0.16420:UINT;
VALx_AnInConf_2 AT %QW0.16424:UINT;
VALx_AnInConf_3 AT %QW0.16428:UINT;
VALx_AnInConf_4 AT %QW0.16432:UINT;
VALx_AnInConf_5 AT %QW0.16436:UINT;
VALx_AnInConf_6 AT %QW0.16440:UINT;
VALx_AnInConf_7 AT %QW0.16444:UINT;
VALx_AnInConf_8 AT %QW0.16448:UINT;
VALx_AnInConf_9 AT %QW0.16452:UINT;
VALx_AnInConf_10 AT %QW0.16456:UINT;
VALx_AnInConf_11 AT %QW0.16460:UINT;
VALx_AnInConf_12 AT %QW0.16464:UINT;
VALx_AnInFltr_1 AT %QW0.16468:UINT;
VALx_AnInFltr_2 AT %QW0.16472:UINT;
VALx_AnInFltr_3 AT %QW0.16476:UINT;
VALx_AnInFltr_4 AT %QW0.16480:UINT;
VALx_AnInFltr_5 AT %QW0.16484:UINT;
VALx_AnInFltr_6 AT %QW0.16488:UINT;
VALx_AnInFltr_7 AT %QW0.16492:UINT;
VALx_AnInFltr_8 AT %QW0.16496:UINT;
VALx_AnInFltr_9 AT %QW0.16500:UINT;
VALx_AnInFltr_10 AT %QW0.16504:UINT;
VALx_AnInFltr_11 AT %QW0.16508:UINT;
VALx_AnInFltr_12 AT %QW0.16512:UINT;
RESx_AnIn_1 AT %IW0.16516:INT;
RESx_AnIn_2 AT %IW0.16520:INT;
RESx_AnIn_3 AT %IW0.16524:INT;
RESx_AnIn_4 AT %IW0.16528:INT;
RESx_AnIn_5 AT %IW0.16532:INT;
RESx_AnIn_6 AT %IW0.16536:INT;
RESx_AnIn_7 AT %IW0.16540:INT;
RESx_AnIn_8 AT %IW0.16544:INT;
RESx_AnIn_9 AT %IW0.16548:INT;
RESx_AnIn_10 AT %IW0.16552:INT;
RESx_AnIn_11 AT %IW0.16556:INT;
RESx_AnIn_12 AT %IW0.16560:INT;
RESx_AnInStts_1 AT %IW0.16564:INT;
RESx_AnInStts_2 AT %IW0.16568:INT;
RESx_AnInStts_3 AT %IW0.16572:INT;
RESx_AnInStts_4 AT %IW0.16576:INT;
RESx_AnInStts_5 AT %IW0.16580:INT;
RESx_AnInStts_6 AT %IW0.16584:INT;
RESx_AnInStts_7 AT %IW0.16588:INT;
RESx_AnInStts_8 AT %IW0.16592:INT;
RESx_AnInStts_9 AT %IW0.16596:INT;
RESx_AnInStts_10 AT %IW0.16600:INT;
RESx_AnInStts_11 AT %IW0.16604:INT;
RESx_AnInStts_12 AT %IW0.16608:INT;
TSTx_AnOut_1 AT %QX0.16612.0:BOOL;
TSTx_AnOut_2 AT %QX0.16616.0:BOOL;
TSTx_AnOut_3 AT %QX0.16620.0:BOOL;
TSTx_AnOut_4 AT %QX0.16624.0:BOOL;
VALx_AnOut_1 AT %QW0.16628:INT;
VALx_AnOut_2 AT %QW0.16632:INT;
VALx_AnOut_3 AT %QW0.16636:INT;
VALx_AnOut_4 AT %QW0.16640:INT;
VALx_AnOutConf_1 AT %QW0.16644:UINT;
VALx_AnOutConf_2 AT %QW0.16648:UINT;
VALx_AnOutConf_3 AT %QW0.16652:UINT;
VALx_AnOutConf_4 AT %QW0.16656:UINT;
RESx_AnOutStts_1 AT %IW0.16660:INT;
RESx_AnOutStts_2 AT %IW0.16664:INT;
RESx_AnOutStts_3 AT %IW0.16668:INT;
RESx_AnOutStts_4 AT %IW0.16672:INT;
TSTx_Tamb AT %QX0.16676.0:BOOL;
TSTx_RPM AT %QX0.16680.0:BOOL;
TSTx_FWrevision AT %QX0.16684.0:BOOL;
TSTx_HWconfig AT %QX0.16688.0:BOOL;
VALx_Tamb AT %QW0.16692:INT;
VALx_RPM AT %QW0.16696:UINT;
VALx_FWrevision AT %QW0.16700:UINT;
VALx_HWconfig AT %QW0.16704:UINT;
RESx_Tamb AT %IW0.16708:INT;
RESx_RPM AT %IW0.16712:UINT;
RESx_FWrevision AT %IW0.16716:UINT;
RESx_HWconfig AT %IW0.16720:UINT;
TSTx_RTUS_WR AT %QX0.16724.0:BOOL;
TSTx_RTUS_RD AT %QX0.16728.0:BOOL;
TSTx_RTU1_WR AT %QX0.16732.0:BOOL;
TSTx_RTU1_RD AT %QX0.16736.0:BOOL;
TSTx_RTU3_WR AT %QX0.16740.0:BOOL;
TSTx_RTU3_RD AT %QX0.16744.0:BOOL;
TSTx_CAN1_WR AT %QX0.16748.0:BOOL;
TSTx_CAN1_RD AT %QX0.16752.0:BOOL;
VALx_RTUS_WR AT %QX0.16756.0:BOOL;
VALx_RTUS_RD AT %QX0.16760.0:BOOL;
VALx_RTU1_WR AT %QX0.16764.0:BOOL;
VALx_RTU1_RD AT %QX0.16768.0:BOOL;
VALx_RTU3_WR AT %QX0.16772.0:BOOL;
VALx_RTU3_RD AT %QX0.16776.0:BOOL;
VALx_CAN1_WR AT %QX0.16780.0:BOOL;
VALx_CAN1_RD AT %QX0.16784.0:BOOL;
RESx_RTUS_WR AT %QX0.16788.0:BOOL;
RESx_RTUS_RD AT %QX0.16792.0:BOOL;
RESx_RTU1_WR AT %QX0.16796.0:BOOL;
RESx_RTU1_RD AT %QX0.16800.0:BOOL;
RESx_RTU3_WR AT %QX0.16804.0:BOOL;
RESx_RTU3_RD AT %QX0.16808.0:BOOL;
RESx_CAN1_WR AT %QX0.16812.0:BOOL;
RESx_CAN1_RD AT %QX0.16816.0:BOOL;
TESTx_STATUS AT %IW0.16820:UINT;
RTU0_TYPE_PORT AT %ID0.20000:UDINT;
RTU0_BAUDRATE AT %ID0.20004:UDINT;
RTU0_STATUS AT %ID0.20008:UDINT;
RTU0_READS AT %ID0.20012:UDINT;
RTU0_WRITES AT %ID0.20016:UDINT;
RTU0_TIMEOUTS AT %ID0.20020:UDINT;
RTU0_COMM_ERRORS AT %ID0.20024:UDINT;
RTU0_LAST_ERROR AT %ID0.20028:UDINT;
RTU0_WRITE_QUEUE AT %ID0.20032:UDINT;
RTU0_READ_QUEUE AT %ID0.20036:UDINT;
RTU1_TYPE_PORT AT %ID0.20040:UDINT;
RTU1_BAUDRATE AT %ID0.20044:UDINT;
RTU1_STATUS AT %ID0.20048:UDINT;
RTU1_READS AT %ID0.20052:UDINT;
RTU1_WRITES AT %ID0.20056:UDINT;
RTU1_TIMEOUTS AT %ID0.20060:UDINT;
RTU1_COMM_ERRORS AT %ID0.20064:UDINT;
RTU1_LAST_ERROR AT %ID0.20068:UDINT;
RTU1_WRITE_QUEUE AT %ID0.20072:UDINT;
RTU1_READ_QUEUE AT %ID0.20076:UDINT;
RTU3_TYPE_PORT AT %ID0.20080:UDINT;
RTU3_BAUDRATE AT %ID0.20084:UDINT;
RTU3_STATUS AT %ID0.20088:UDINT;
RTU3_READS AT %ID0.20092:UDINT;
RTU3_WRITES AT %ID0.20096:UDINT;
RTU3_TIMEOUTS AT %ID0.20100:UDINT;
RTU3_COMM_ERRORS AT %ID0.20104:UDINT;
RTU3_LAST_ERROR AT %ID0.20108:UDINT;
RTU3_WRITE_QUEUE AT %ID0.20112:UDINT;
RTU3_READ_QUEUE AT %ID0.20116:UDINT;
CAN0_TYPE_PORT AT %ID0.20120:UDINT;
CAN0_BAUDRATE AT %ID0.20124:UDINT;
CAN0_STATUS AT %ID0.20128:UDINT;
CAN0_READS AT %ID0.20132:UDINT;
CAN0_WRITES AT %ID0.20136:UDINT;
CAN0_TIMEOUTS AT %ID0.20140:UDINT;
CAN0_COMM_ERRORS AT %ID0.20144:UDINT;
CAN0_LAST_ERROR AT %ID0.20148:UDINT;
CAN0_WRITE_QUEUE AT %ID0.20152:UDINT;
CAN0_READ_QUEUE AT %ID0.20156:UDINT;
CAN1_TYPE_PORT AT %ID0.20160:UDINT;
CAN1_BAUDRATE AT %ID0.20164:UDINT;
CAN1_STATUS AT %ID0.20168:UDINT;
CAN1_READS AT %ID0.20172:UDINT;
CAN1_WRITES AT %ID0.20176:UDINT;
CAN1_TIMEOUTS AT %ID0.20180:UDINT;
CAN1_COMM_ERRORS AT %ID0.20184:UDINT;
CAN1_LAST_ERROR AT %ID0.20188:UDINT;
CAN1_WRITE_QUEUE AT %ID0.20192:UDINT;
CAN1_READ_QUEUE AT %ID0.20196:UDINT;
TCPS_TYPE_PORT AT %ID0.20200:UDINT;
TCPS_IP_ADDRESS AT %ID0.20204:UDINT;
TCPS_STATUS AT %ID0.20208:UDINT;
TCPS_READS AT %ID0.20212:UDINT;
TCPS_WRITES AT %ID0.20216:UDINT;
TCPS_TIMEOUTS AT %ID0.20220:UDINT;
TCPS_COMM_ERRORS AT %ID0.20224:UDINT;
TCPS_LAST_ERROR AT %ID0.20228:UDINT;
TCPS_WRITE_QUEUE AT %ID0.20232:UDINT;
TCPS_READ_QUEUE AT %ID0.20236:UDINT;
TCP0_TYPE_PORT AT %ID0.20240:UDINT;
TCP0_IP_ADDRESS AT %ID0.20244:UDINT;
TCP0_STATUS AT %ID0.20248:UDINT;
TCP0_READS AT %ID0.20252:UDINT;
TCP0_WRITES AT %ID0.20256:UDINT;
TCP0_TIMEOUTS AT %ID0.20260:UDINT;
TCP0_COMM_ERRORS AT %ID0.20264:UDINT;
TCP0_LAST_ERROR AT %ID0.20268:UDINT;
TCP0_WRITE_QUEUE AT %ID0.20272:UDINT;
TCP0_READ_QUEUE AT %ID0.20276:UDINT;
TCP1_TYPE_PORT AT %ID0.20280:UDINT;
TCP1_IP_ADDRESS AT %ID0.20284:UDINT;
TCP1_STATUS AT %ID0.20288:UDINT;
TCP1_READS AT %ID0.20292:UDINT;
TCP1_WRITES AT %ID0.20296:UDINT;
TCP1_TIMEOUTS AT %ID0.20300:UDINT;
TCP1_COMM_ERRORS AT %ID0.20304:UDINT;
TCP1_LAST_ERROR AT %ID0.20308:UDINT;
TCP1_WRITE_QUEUE AT %ID0.20312:UDINT;
TCP1_READ_QUEUE AT %ID0.20316:UDINT;
TCP2_TYPE_PORT AT %ID0.20320:UDINT;
TCP2_IP_ADDRESS AT %ID0.20324:UDINT;
TCP2_STATUS AT %ID0.20328:UDINT;
TCP2_READS AT %ID0.20332:UDINT;
TCP2_WRITES AT %ID0.20336:UDINT;
TCP2_TIMEOUTS AT %ID0.20340:UDINT;
TCP2_COMM_ERRORS AT %ID0.20344:UDINT;
TCP2_LAST_ERROR AT %ID0.20348:UDINT;
TCP2_WRITE_QUEUE AT %ID0.20352:UDINT;
TCP2_READ_QUEUE AT %ID0.20356:UDINT;
TCP3_TYPE_PORT AT %ID0.20360:UDINT;
TCP3_IP_ADDRESS AT %ID0.20364:UDINT;
TCP3_STATUS AT %ID0.20368:UDINT;
TCP3_READS AT %ID0.20372:UDINT;
TCP3_WRITES AT %ID0.20376:UDINT;
TCP3_TIMEOUTS AT %ID0.20380:UDINT;
TCP3_COMM_ERRORS AT %ID0.20384:UDINT;
TCP3_LAST_ERROR AT %ID0.20388:UDINT;
TCP3_WRITE_QUEUE AT %ID0.20392:UDINT;
TCP3_READ_QUEUE AT %ID0.20396:UDINT;
TCP4_TYPE_PORT AT %ID0.20400:UDINT;
TCP4_IP_ADDRESS AT %ID0.20404:UDINT;
TCP4_STATUS AT %ID0.20408:UDINT;
TCP4_READS AT %ID0.20412:UDINT;
TCP4_WRITES AT %ID0.20416:UDINT;
TCP4_TIMEOUTS AT %ID0.20420:UDINT;
TCP4_COMM_ERRORS AT %ID0.20424:UDINT;
TCP4_LAST_ERROR AT %ID0.20428:UDINT;
TCP4_WRITE_QUEUE AT %ID0.20432:UDINT;
TCP4_READ_QUEUE AT %ID0.20436:UDINT;
TCP5_TYPE_PORT AT %ID0.20440:UDINT;
TCP5_IP_ADDRESS AT %ID0.20444:UDINT;
TCP5_STATUS AT %ID0.20448:UDINT;
TCP5_READS AT %ID0.20452:UDINT;
TCP5_WRITES AT %ID0.20456:UDINT;
TCP5_TIMEOUTS AT %ID0.20460:UDINT;
TCP5_COMM_ERRORS AT %ID0.20464:UDINT;
TCP5_LAST_ERROR AT %ID0.20468:UDINT;
TCP5_WRITE_QUEUE AT %ID0.20472:UDINT;
TCP5_READ_QUEUE AT %ID0.20476:UDINT;
TCP6_TYPE_PORT AT %ID0.20480:UDINT;
TCP6_IP_ADDRESS AT %ID0.20484:UDINT;
TCP6_STATUS AT %ID0.20488:UDINT;
TCP6_READS AT %ID0.20492:UDINT;
TCP6_WRITES AT %ID0.20496:UDINT;
TCP6_TIMEOUTS AT %ID0.20500:UDINT;
TCP6_COMM_ERRORS AT %ID0.20504:UDINT;
TCP6_LAST_ERROR AT %ID0.20508:UDINT;
TCP6_WRITE_QUEUE AT %ID0.20512:UDINT;
TCP6_READ_QUEUE AT %ID0.20516:UDINT;
TCP7_TYPE_PORT AT %ID0.20520:UDINT;
TCP7_IP_ADDRESS AT %ID0.20524:UDINT;
TCP7_STATUS AT %ID0.20528:UDINT;
TCP7_READS AT %ID0.20532:UDINT;
TCP7_WRITES AT %ID0.20536:UDINT;
TCP7_TIMEOUTS AT %ID0.20540:UDINT;
TCP7_COMM_ERRORS AT %ID0.20544:UDINT;
TCP7_LAST_ERROR AT %ID0.20548:UDINT;
TCP7_WRITE_QUEUE AT %ID0.20552:UDINT;
TCP7_READ_QUEUE AT %ID0.20556:UDINT;
TCP8_TYPE_PORT AT %ID0.20560:UDINT;
TCP8_IP_ADDRESS AT %ID0.20564:UDINT;
TCP8_STATUS AT %ID0.20568:UDINT;
TCP8_READS AT %ID0.20572:UDINT;
TCP8_WRITES AT %ID0.20576:UDINT;
TCP8_TIMEOUTS AT %ID0.20580:UDINT;
TCP8_COMM_ERRORS AT %ID0.20584:UDINT;
TCP8_LAST_ERROR AT %ID0.20588:UDINT;
TCP8_WRITE_QUEUE AT %ID0.20592:UDINT;
TCP8_READ_QUEUE AT %ID0.20596:UDINT;
TCP9_TYPE_PORT AT %ID0.20600:UDINT;
TCP9_IP_ADDRESS AT %ID0.20604:UDINT;
TCP9_STATUS AT %ID0.20608:UDINT;
TCP9_READS AT %ID0.20612:UDINT;
TCP9_WRITES AT %ID0.20616:UDINT;
TCP9_TIMEOUTS AT %ID0.20620:UDINT;
TCP9_COMM_ERRORS AT %ID0.20624:UDINT;
TCP9_LAST_ERROR AT %ID0.20628:UDINT;
TCP9_WRITE_QUEUE AT %ID0.20632:UDINT;
TCP9_READ_QUEUE AT %ID0.20636:UDINT;
NODE_01_DEV_NODE AT %ID0.20688:UDINT;
NODE_01_STATUS AT %ID0.20692:UDINT;
NODE_02_DEV_NODE AT %ID0.20696:UDINT;
NODE_02_STATUS AT %ID0.20700:UDINT;
NODE_03_DEV_NODE AT %ID0.20704:UDINT;
NODE_03_STATUS AT %ID0.20708:UDINT;
NODE_04_DEV_NODE AT %ID0.20712:UDINT;
NODE_04_STATUS AT %ID0.20716:UDINT;
NODE_05_DEV_NODE AT %ID0.20720:UDINT;
NODE_05_STATUS AT %ID0.20724:UDINT;
NODE_06_DEV_NODE AT %ID0.20728:UDINT;
NODE_06_STATUS AT %ID0.20732:UDINT;
NODE_07_DEV_NODE AT %ID0.20736:UDINT;
NODE_07_STATUS AT %ID0.20740:UDINT;
NODE_08_DEV_NODE AT %ID0.20744:UDINT;
NODE_08_STATUS AT %ID0.20748:UDINT;
NODE_09_DEV_NODE AT %ID0.20752:UDINT;
NODE_09_STATUS AT %ID0.20756:UDINT;
NODE_10_DEV_NODE AT %ID0.20760:UDINT;
NODE_10_STATUS AT %ID0.20764:UDINT;
NODE_11_DEV_NODE AT %ID0.20768:UDINT;
NODE_11_STATUS AT %ID0.20772:UDINT;
NODE_12_DEV_NODE AT %ID0.20776:UDINT;
NODE_12_STATUS AT %ID0.20780:UDINT;
NODE_13_DEV_NODE AT %ID0.20784:UDINT;
NODE_13_STATUS AT %ID0.20788:UDINT;
NODE_14_DEV_NODE AT %ID0.20792:UDINT;
NODE_14_STATUS AT %ID0.20796:UDINT;
NODE_15_DEV_NODE AT %ID0.20800:UDINT;
NODE_15_STATUS AT %ID0.20804:UDINT;
NODE_16_DEV_NODE AT %ID0.20808:UDINT;
NODE_16_STATUS AT %ID0.20812:UDINT;
PLC_FWrevision AT %IW0.21200:UINT;
PLC_HWconfig AT %IW0.21204:UINT;
PLC_DigDir_1 AT %QX0.21208.0:BOOL;
PLC_DigDir_2 AT %QX0.21212.0:BOOL;
PLC_DigDir_3 AT %QX0.21216.0:BOOL;
PLC_DigDir_4 AT %QX0.21220.0:BOOL;
PLC_DigDir_5 AT %QX0.21224.0:BOOL;
PLC_DigDir_6 AT %QX0.21228.0:BOOL;
PLC_DigDir_7 AT %QX0.21232.0:BOOL;
PLC_DigDir_8 AT %QX0.21236.0:BOOL;
PLC_AnInConf_1 AT %QW0.21240:UINT;
PLC_AnInConf_2 AT %QW0.21244:UINT;
PLC_AnOutConf_1 AT %QW0.21248:UINT;
PLC_AnOutConf_2 AT %QW0.21252:UINT;
PLC_AnOutConf_3 AT %QW0.21256:UINT;
PLC_AnOutConf_4 AT %QW0.21260:UINT;
PLC_DigIn_1 AT %IX0.21264.0:BOOL;
PLC_DigIn_2 AT %IX0.21268.0:BOOL;
PLC_DigIn_3 AT %IX0.21272.0:BOOL;
PLC_DigIn_4 AT %IX0.21276.0:BOOL;
PLC_DigIn_5 AT %IX0.21280.0:BOOL;
PLC_DigIn_6 AT %IX0.21284.0:BOOL;
PLC_DigIn_7 AT %IX0.21288.0:BOOL;
PLC_DigIn_8 AT %IX0.21292.0:BOOL;
PLC_DigIn_9 AT %IX0.21296.0:BOOL;
PLC_DigIn_10 AT %IX0.21300.0:BOOL;
PLC_DigIn_11 AT %IX0.21304.0:BOOL;
PLC_DigIn_12 AT %IX0.21308.0:BOOL;
PLC_AnIn_1 AT %IW0.21312:INT;
PLC_AnIn_2 AT %IW0.21316:INT;
PLC_Reserved_1 AT %IW0.21320:INT;
PLC_Reserved_2 AT %IW0.21324:INT;
PLC_Reserved_3 AT %IW0.21328:INT;
PLC_Tamb AT %IW0.21332:INT;
PLC_Encoder AT %ID0.21336:DINT;
PLC_Capture AT %ID0.21340:UDINT;
PLC_DigOut_1 AT %QX0.21344.0:BOOL;
PLC_DigOut_2 AT %QX0.21348.0:BOOL;
PLC_DigOut_3 AT %QX0.21352.0:BOOL;
PLC_DigOut_4 AT %QX0.21356.0:BOOL;
PLC_DigOut_5 AT %QX0.21360.0:BOOL;
PLC_DigOut_6 AT %QX0.21364.0:BOOL;
PLC_DigOut_7 AT %QX0.21368.0:BOOL;
PLC_DigOut_8 AT %QX0.21372.0:BOOL;
PLC_AnOut_1 AT %QW0.21376:INT;
PLC_AnOut_2 AT %QW0.21380:INT;
PLC_AnOut_3 AT %QW0.21384:INT;
PLC_AnOut_4 AT %QW0.21388:INT;
PLC_EncoderStart AT %QW0.21392:UINT;
PLC_EncoderReset AT %QW0.21396:UINT;
PLC_Heartbeat AT %IW0.21400:UINT;
PLC_StatusReg AT %IW0.21404:UINT;
PLC_AnIn1Filter AT %QW0.21408:UINT;
PLC_AnIn2Filter AT %QW0.21412:UINT;
PLC_time AT %ID0.21560:REAL;
PLC_timeMin AT %ID0.21564:REAL;
PLC_timeMax AT %ID0.21568:REAL;
PLC_timeWin AT %QD0.21572:REAL;
PLC_Version AT %IW0.21576:UINT;
PLC_EngineStatus AT %IW0.21580:UINT;
PLC_ResetValues AT %QX0.21584.0:BOOL;
PLC_buzzerOn AT %QX0.21588.0:BOOL;
END_VAR

(* ---- Resource1.gvl ---- *)
(* Global variable file *)
VAR_GLOBAL

END_VAR

(* ---- AllTestedAreOK.st ---- *)
(*[[
]]*)
FUNCTION AllTestedAreOK : BOOL
#import "Crosstable.gvl"
VAR
	retval : BOOL := TRUE;
END_VAR

	if TST_DigIn_1  then retval := retval and OK_DigIn_1;  end_if;
	if TST_DigIn_2  then retval := retval and OK_DigIn_2;  end_if;
	if TST_DigIn_3  then retval := retval and OK_DigIn_3;  end_if;
	if TST_DigIn_4  then retval := retval and OK_DigIn_4;  end_if;
	if TST_DigIn_5  then retval := retval and OK_DigIn_5;  end_if;
	if TST_DigIn_6  then retval := retval and OK_DigIn_6;  end_if;
	if TST_DigIn_7  then retval := retval and OK_DigIn_7;  end_if;
	if TST_DigIn_8  then retval := retval and OK_DigIn_8;  end_if;
	if TST_DigIn_9  then retval := retval and OK_DigIn_9;  end_if;
	if TST_DigIn_10 then retval := retval and OK_DigIn_10; end_if;
	if TST_DigIn_11 then retval := retval and OK_DigIn_11; end_if;
	if TST_DigIn_12 then retval := retval and OK_DigIn_12; end_if;
	if TST_DigIn_13 then retval := retval and OK_DigIn_13; end_if;
	if TST_DigIn_14 then retval := retval and OK_DigIn_14; end_if;
	if TST_DigIn_15 then retval := retval and OK_DigIn_15; end_if;
	if TST_DigIn_16 then retval := retval and OK_DigIn_16; end_if;

	if TST_DigOut_1  then retval := retval and OK_DigOut_1;  end_if;
	if TST_DigOut_2  then retval := retval and OK_DigOut_2;  end_if;
	if TST_DigOut_3  then retval := retval and OK_DigOut_3;  end_if;
	if TST_DigOut_4  then retval := retval and OK_DigOut_4;  end_if;
	if TST_DigOut_5  then retval := retval and OK_DigOut_5;  end_if;
	if TST_DigOut_6  then retval := retval and OK_DigOut_6;  end_if;
	if TST_DigOut_7  then retval := retval and OK_DigOut_7;  end_if;
	if TST_DigOut_8  then retval := retval and OK_DigOut_8;  end_if;
	if TST_DigOut_9  then retval := retval and OK_DigOut_9;  end_if;
	if TST_DigOut_10 then retval := retval and OK_DigOut_10; end_if;
	if TST_DigOut_11 then retval := retval and OK_DigOut_11; end_if;
	if TST_DigOut_12 then retval := retval and OK_DigOut_12; end_if;
	if TST_DigOut_13 then retval := retval and OK_DigOut_13; end_if;
	if TST_DigOut_14 then retval := retval and OK_DigOut_14; end_if;
	if TST_DigOut_15 then retval := retval and OK_DigOut_15; end_if;
	if TST_DigOut_16 then retval := retval and OK_DigOut_16; end_if;

	if TST_AnIn_1  then retval := retval and OK_AnIn_1;  end_if;
	if TST_AnIn_2  then retval := retval and OK_AnIn_2;  end_if;
	if TST_AnIn_3  then retval := retval and OK_AnIn_3;  end_if;
	if TST_AnIn_4  then retval := retval and OK_AnIn_4;  end_if;

	if TST_AnIn_5  then retval := retval and OK_AnIn_5;  end_if;
	if TST_AnIn_6  then retval := retval and OK_AnIn_6;  end_if;
	if TST_AnIn_7  then retval := retval and OK_AnIn_7;  end_if;
	if TST_AnIn_8  then retval := retval and OK_AnIn_8;  end_if;
	if TST_AnIn_9  then retval := retval and OK_AnIn_9;  end_if;
	if TST_AnIn_10 then retval := retval and OK_AnIn_10;  end_if;
	if TST_AnIn_11 then retval := retval and OK_AnIn_11;  end_if;
	if TST_AnIn_12 then retval := retval and OK_AnIn_12;  end_if;

	if TST_AnOut_1  then retval := retval and OK_AnOut_1;  end_if;
	if TST_AnOut_2  then retval := retval and OK_AnOut_2;  end_if;
	if TST_AnOut_3  then retval := retval and OK_AnOut_3;  end_if;
	if TST_AnOut_4  then retval := retval and OK_AnOut_4;  end_if;

	if TST_Tamb  then retval := retval and OK_Tamb;  end_if;
	if TST_RPM   then retval := retval and OK_RPM;  end_if;

	if TST_VCC_set  then retval := retval and OK_VCC_set;  end_if;
	if TST_mA_max  then retval := retval and OK_mA_max;  end_if;

	if TST_VCC_fbk  then retval := retval and OK_VCC_fbk;  end_if;
	if TST_mA_fbk  then retval := retval and OK_mA_fbk;  end_if;

	if TST_FWrevision  then retval := retval and OK_FWrevision; end_if;
	if TST_HWconfig  then retval := retval and OK_HWconfig;  end_if;

	if TST_RTU1_WR  then retval := retval and OK_RTU1_WR; end_if;
	if TST_RTU1_RD  then retval := retval and OK_RTU1_RD; end_if;
	if TST_RTU3_WR  then retval := retval and OK_RTU3_WR; end_if;
	if TST_RTU3_RD  then retval := retval and OK_RTU3_RD; end_if;

	AllTestedAreOK := retval;
END_FUNCTION

(* ---- Check_AnIn.st ---- *)
(*[[
]]*)
FUNCTION Check_AnIn
#import "Crosstable.gvl"
VAR_INPUT
END_VAR
VAR
	Tolleranza : INT := 1; (* 0.001 *)
END_VAR

	(* Get results *)
	if TST_AnIn_1  then RES_AnIn_1  := RESx_AnIn_1;  end_if;
	if TST_AnIn_2  then RES_AnIn_2  := RESx_AnIn_2;  end_if;
	if TST_AnIn_3  then RES_AnIn_3  := RESx_AnIn_3;  end_if;
	if TST_AnIn_4  then RES_AnIn_4  := RESx_AnIn_4;  end_if;

	if TST_AnIn_5  then RES_AnIn_5  := RESx_AnIn_5;  end_if;
	if TST_AnIn_6  then RES_AnIn_6  := RESx_AnIn_6;  end_if;
	if TST_AnIn_7  then RES_AnIn_7  := RESx_AnIn_7;  end_if;
	if TST_AnIn_8  then RES_AnIn_8  := RESx_AnIn_8;  end_if;
	if TST_AnIn_9  then RES_AnIn_9  := RESx_AnIn_9;  end_if;
	if TST_AnIn_10 then RES_AnIn_10 := RESx_AnIn_10;  end_if;
	if TST_AnIn_11 then RES_AnIn_11 := RESx_AnIn_11;  end_if;
	if TST_AnIn_12 then RES_AnIn_12 := RESx_AnIn_12;  end_if;

	(* Check values *)
	if TST_AnIn_1  then OK_AnIn_1  := abs(RES_AnIn_1  - VAL_AnIn_1 ) < Tolleranza; end_if;
	if TST_AnIn_2  then OK_AnIn_2  := abs(RES_AnIn_2  - VAL_AnIn_2 ) < Tolleranza; end_if;
	if TST_AnIn_3  then OK_AnIn_3  := abs(RES_AnIn_3  - VAL_AnIn_3 ) < Tolleranza; end_if;
	if TST_AnIn_4  then OK_AnIn_4  := abs(RES_AnIn_4  - VAL_AnIn_4 ) < Tolleranza; end_if;

	if TST_AnIn_5  then OK_AnIn_5  := abs(RES_AnIn_5  - VAL_AnIn_5 ) < Tolleranza; end_if;
	if TST_AnIn_6  then OK_AnIn_6  := abs(RES_AnIn_6  - VAL_AnIn_6 ) < Tolleranza; end_if;
	if TST_AnIn_7  then OK_AnIn_7  := abs(RES_AnIn_7  - VAL_AnIn_7 ) < Tolleranza; end_if;
	if TST_AnIn_8  then OK_AnIn_8  := abs(RES_AnIn_8  - VAL_AnIn_8 ) < Tolleranza; end_if;
	if TST_AnIn_9  then OK_AnIn_9  := abs(RES_AnIn_9  - VAL_AnIn_9 ) < Tolleranza; end_if;
	if TST_AnIn_10 then OK_AnIn_10 := abs(RES_AnIn_10 - VAL_AnIn_10) < Tolleranza; end_if;
	if TST_AnIn_11 then OK_AnIn_11 := abs(RES_AnIn_11 - VAL_AnIn_11) < Tolleranza; end_if;
	if TST_AnIn_12 then OK_AnIn_12 := abs(RES_AnIn_12 - VAL_AnIn_12) < Tolleranza; end_if;

END_FUNCTION

(* ---- Check_AnOut.st ---- *)
(*[[
]]*)
FUNCTION Check_AnOut
#import "Crosstable.gvl"
VAR_INPUT
END_VAR
VAR
	Tolleranza : INT := 1; (* 0.01 *)
END_VAR

	(* Get results *)
	if TST_AnOut_1  then RES_AnOut_1 := RES2_AnIn_1;  end_if;
	if TST_AnOut_2  then RES_AnOut_2 := RES2_AnIn_2;  end_if;
	if TST_AnOut_3  then RES_AnOut_3 := RTU_AnIn_1;  end_if;
	if TST_AnOut_4  then RES_AnOut_4 := RTU_AnIn_2;  end_if;

	(* Check values *)
	if TST_AnOut_1  then OK_AnOut_1 := abs(RES_AnOut_1 - VAL_AnOut_1) < Tolleranza; end_if;
	if TST_AnOut_2  then OK_AnOut_2 := abs(RES_AnOut_2 - VAL_AnOut_2) < Tolleranza; end_if;
	if TST_AnOut_3  then OK_AnOut_3 := abs(RES_AnOut_3 - VAL_AnOut_3) < Tolleranza; end_if;
	if TST_AnOut_4  then OK_AnOut_4 := abs(RES_AnOut_4 - VAL_AnOut_4) < Tolleranza; end_if;

END_FUNCTION

(* ---- Check_DigIn.st ---- *)
(*[[
]]*)
FUNCTION Check_DigIn
#import "Crosstable.gvl"
VAR_INPUT
END_VAR

	(* Get results *)
	if TST_DigIn_1  then RES_DigIn_1 := RESx_DigIn_1;  end_if;
	if TST_DigIn_2  then RES_DigIn_2 := RESx_DigIn_2;  end_if;
	if TST_DigIn_3  then RES_DigIn_3 := RESx_DigIn_3;  end_if;
	if TST_DigIn_4  then RES_DigIn_4 := RESx_DigIn_4;  end_if;
	if TST_DigIn_5  then RES_DigIn_5 := RESx_DigIn_5;  end_if;
	if TST_DigIn_6  then RES_DigIn_6 := RESx_DigIn_6;  end_if;
	if TST_DigIn_7  then RES_DigIn_7 := RESx_DigIn_7;  end_if;
	if TST_DigIn_8  then RES_DigIn_8 := RESx_DigIn_8;  end_if;
	if TST_DigIn_9  then RES_DigIn_9 := RESx_DigIn_9;  end_if;
	if TST_DigIn_10 then RES_DigIn_10:= RESx_DigIn_10; end_if;
	if TST_DigIn_11 then RES_DigIn_11:= RESx_DigIn_11; end_if;
	if TST_DigIn_12 then RES_DigIn_12:= RESx_DigIn_12; end_if;
	if TST_DigIn_13 then RES_DigIn_13:= RESx_DigIn_13; end_if;
	if TST_DigIn_14 then RES_DigIn_14:= RESx_DigIn_14; end_if;
	if TST_DigIn_15 then RES_DigIn_15:= RESx_DigIn_15; end_if;
	if TST_DigIn_16 then RES_DigIn_16:= RESx_DigIn_16; end_if;

	(* Check values *)
	if TST_DigIn_1  then OK_DigIn_1 := (RES_DigIn_1 = VAL_DigIn_1);  end_if;
	if TST_DigIn_2  then OK_DigIn_2 := (RES_DigIn_2 = VAL_DigIn_2);  end_if;
	if TST_DigIn_3  then OK_DigIn_3 := (RES_DigIn_3 = VAL_DigIn_3);  end_if;
	if TST_DigIn_4  then OK_DigIn_4 := (RES_DigIn_4 = VAL_DigIn_4);  end_if;
	if TST_DigIn_5  then OK_DigIn_5 := (RES_DigIn_5 = VAL_DigIn_5);  end_if;
	if TST_DigIn_6  then OK_DigIn_6 := (RES_DigIn_6 = VAL_DigIn_6);  end_if;
	if TST_DigIn_7  then OK_DigIn_7 := (RES_DigIn_7 = VAL_DigIn_7);  end_if;
	if TST_DigIn_8  then OK_DigIn_8 := (RES_DigIn_8 = VAL_DigIn_8);  end_if;
	if TST_DigIn_9  then OK_DigIn_9 := (RES_DigIn_9 = VAL_DigIn_9);  end_if;
	if TST_DigIn_10 then OK_DigIn_10:= (RES_DigIn_10 = VAL_DigIn_10); end_if;
	if TST_DigIn_11 then OK_DigIn_11:= (RES_DigIn_11 = VAL_DigIn_11); end_if;
	if TST_DigIn_12 then OK_DigIn_12:= (RES_DigIn_12 = VAL_DigIn_12); end_if;
	if TST_DigIn_13 then OK_DigIn_13:= (RES_DigIn_13 = VAL_DigIn_13); end_if;
	if TST_DigIn_14 then OK_DigIn_14:= (RES_DigIn_14 = VAL_DigIn_14); end_if;
	if TST_DigIn_15 then OK_DigIn_15:= (RES_DigIn_15 = VAL_DigIn_15); end_if;
	if TST_DigIn_16 then OK_DigIn_16:= (RES_DigIn_16 = VAL_DigIn_16); end_if;

END_FUNCTION

(* ---- Check_DigOut.st ---- *)
(*[[
]]*)
FUNCTION Check_DigOut
#import "Crosstable.gvl"
VAR_INPUT
END_VAR

	(* Get results *)
	if TST_DigOut_1  then RES_DigOut_1 := RTU_DigIn_1;  end_if;
	if TST_DigOut_2  then RES_DigOut_2 := RTU_DigIn_2;  end_if;
	if TST_DigOut_3  then RES_DigOut_3 := RTU_DigIn_3;  end_if;
	if TST_DigOut_4  then RES_DigOut_4 := RTU_DigIn_4;  end_if;
	if TST_DigOut_5  then RES_DigOut_5 := RTU_DigIn_5;  end_if;
	if TST_DigOut_6  then RES_DigOut_6 := RTU_DigIn_6;  end_if;
	if TST_DigOut_7  then RES_DigOut_7 := RTU_DigIn_7;  end_if;
	if TST_DigOut_8  then RES_DigOut_8 := RTU_DigIn_8;  end_if;
	if TST_DigOut_9  then RES_DigOut_9 := RTU_DigIn_9;  end_if;
	if TST_DigOut_10 then RES_DigOut_10:= RTU_DigIn_10; end_if;
	if TST_DigOut_11 then RES_DigOut_11:= RTU_DigIn_11; end_if;
	if TST_DigOut_12 then RES_DigOut_12:= RTU_DigIn_12; end_if;
	if TST_DigOut_13 then RES_DigOut_13:= RTU_DigIn_13; end_if;
	if TST_DigOut_14 then RES_DigOut_14:= RTU_DigIn_14; end_if;
	if TST_DigOut_15 then RES_DigOut_15:= RTU_DigIn_15; end_if;
	if TST_DigOut_16 then RES_DigOut_16:= RTU_DigIn_16; end_if;

	(* Check values *)
	if TST_DigOut_1  then OK_DigOut_1 := (RES_DigOut_1 = VAL_DigOut_1);  end_if;
	if TST_DigOut_2  then OK_DigOut_2 := (RES_DigOut_2 = VAL_DigOut_2);  end_if;
	if TST_DigOut_3  then OK_DigOut_3 := (RES_DigOut_3 = VAL_DigOut_3);  end_if;
	if TST_DigOut_4  then OK_DigOut_4 := (RES_DigOut_4 = VAL_DigOut_4);  end_if;
	if TST_DigOut_5  then OK_DigOut_5 := (RES_DigOut_5 = VAL_DigOut_5);  end_if;
	if TST_DigOut_6  then OK_DigOut_6 := (RES_DigOut_6 = VAL_DigOut_6);  end_if;
	if TST_DigOut_7  then OK_DigOut_7 := (RES_DigOut_7 = VAL_DigOut_7);  end_if;
	if TST_DigOut_8  then OK_DigOut_8 := (RES_DigOut_8 = VAL_DigOut_8);  end_if;
	if TST_DigOut_9  then OK_DigOut_9 := (RES_DigOut_9 = VAL_DigOut_9);  end_if;
	if TST_DigOut_10 then OK_DigOut_10:= (RES_DigOut_10 = VAL_DigOut_10); end_if;
	if TST_DigOut_11 then OK_DigOut_11:= (RES_DigOut_11 = VAL_DigOut_11); end_if;
	if TST_DigOut_12 then OK_DigOut_12:= (RES_DigOut_12 = VAL_DigOut_12); end_if;
	if TST_DigOut_13 then OK_DigOut_13:= (RES_DigOut_13 = VAL_DigOut_13); end_if;
	if TST_DigOut_14 then OK_DigOut_14:= (RES_DigOut_14 = VAL_DigOut_14); end_if;
	if TST_DigOut_15 then OK_DigOut_15:= (RES_DigOut_15 = VAL_DigOut_15); end_if;
	if TST_DigOut_16 then OK_DigOut_16:= (RES_DigOut_16 = VAL_DigOut_16); end_if;

END_FUNCTION

(* ---- Check_Others.st ---- *)
(*[[
]]*)
FUNCTION Check_Others
#import "Crosstable.gvl"
VAR_INPUT
END_VAR
VAR
	Tolleranza_Tamb_min : INT := 10;
	Tolleranza_RPM : INT := 100;
	Tolleranza_VCC_set : INT := 10; (* 0.01 V *)
	Tolleranza_mA_max : INT := 10; (* 0.01 mA *)
	Tolleranza_VCC_fbk : INT := 100; (* 0.1 V *)
	Tolleranza_mA_fbk : INT := 100; (* 0.1 mA *)
END_VAR

	(* Get results *)
	if TST_Tamb  then RES_Tamb  := RESx_Tamb;  end_if;
	if TST_RPM   then RES_RPM  := RESx_RPM;  end_if;

	if TST_VCC_set  then RES_VCC_set  := PLC_AnOut_3;  end_if;
	if TST_mA_max  then RES_mA_max  := PLC_AnOut_4;  end_if;

	if TST_VCC_fbk  then RES_VCC_fbk  := PLC_AnIn_1;  end_if;
	if TST_mA_fbk  then RES_mA_fbk  := PLC_AnIn_2;  end_if;

	if TST_FWrevision  then RES_FWrevision  := RESx_FWrevision;  end_if;
	if TST_HWconfig  then RES_HWconfig  := RESx_HWconfig;  end_if;

	(* Check values *)
	if TST_Tamb  then OK_Tamb  := (Tolleranza_Tamb_min <= RES_Tamb) and (RES_Tamb < VAL_Tamb ); end_if;
	if TST_RPM  then OK_RPM  := abs(UINT_TO_INT(RES_RPM) - UINT_TO_INT(VAL_RPM) ) < Tolleranza_RPM; end_if;

	if TST_VCC_set  then OK_VCC_set  := abs(RES_VCC_set  - VAL_VCC_set ) < Tolleranza_VCC_set; end_if;
	if TST_mA_max  then OK_mA_max  := abs(RES_mA_max - VAL_mA_max ) < Tolleranza_mA_max; end_if;

	if TST_VCC_fbk  then OK_VCC_fbk  := abs(RES_VCC_fbk  - VAL_VCC_fbk ) < Tolleranza_VCC_fbk; end_if;
	if TST_mA_fbk  then OK_mA_fbk := abs(RES_mA_fbk - VAL_mA_fbk ) < Tolleranza_mA_fbk; end_if;

	if TST_FWrevision  then OK_FWrevision  := (RES_FWrevision  = VAL_FWrevision); end_if;
	if TST_HWconfig  then OK_HWconfig  := (RES_HWconfig = VAL_HWconfig); end_if;

END_FUNCTION

(* ---- CheckAnIn.st ---- *)
(*[[
]]*)
FUNCTION CheckAnIn : BOOL
VAR_INPUT
    res : INT;
    val : INT;
    conf : UINT;
END_VAR

    case conf of
    1: (* 4.000 20.000 mA *)
		CheckAnIn := abs(res  - val ) <= 100; (* 0.10mA *)
	2: (* 0.000 10.000 V *)
		CheckAnIn := abs(res  - val ) <= 100; (* 0.100V *)
	3: (* TCJ 0  600 C*)
		CheckAnIn := abs(res  - val ) <= 10; (* 10 C, 35=25..45 *)
	4: (* TCK 0 1200 C*)
		CheckAnIn := abs(res  - val ) <= 1; (* 1 C *)
	5: (* TCT *)
		CheckAnIn := abs(res  - val ) <= 1; (* 1 C *)
	6: (* PT100E *)
		CheckAnIn := abs(res  - val ) <= 5; (* 5 C, 51=46..54 *)
	7: (* PT100R *)
		CheckAnIn := abs(res  - val ) <= 50; (* 5 C, 510=460..540 *)
	8: (* TCS *)
		CheckAnIn := abs(res  - val ) <= 1; (* 1 C *)
	9: (* TCB *)
		CheckAnIn := abs(res  - val ) <= 1; (* 1 C *)
	10: (* TCR *)
		CheckAnIn := abs(res  - val ) <= 1; (* 1 C *)
    else
    	CheckAnIn := FALSE;
    end_case;

END_FUNCTION

(* ---- CheckAnOut.st ---- *)
(*[[
]]*)
FUNCTION CheckAnOut : BOOL
VAR_INPUT
    res : INT;
    val : INT;
    conf : UINT;
END_VAR

    case conf of
    1: (* 4.00 20.00 mA *)
		CheckAnOut := abs(res  - val ) <= 10; (* 0.10mA *)
	2: (* 0.00 10.00 V *)
		CheckAnOut := abs(res  - val ) <= 10; (* 0.100V *)
	3: (* PWM  0 100 *)
		CheckAnOut := abs(res  - val ) <= 10; (* 10 % *)
    else
    	CheckAnOut := FALSE;
    end_case;

END_FUNCTION

(* ---- CheckOK.st ---- *)
(*[[
]]*)
FUNCTION CheckOK
#import "Crosstable.gvl"
VAR_INPUT
END_VAR
VAR
	Tolleranza_In : INT := 100; (* 20mV = 2 * 10mV *)
	Tolleranza_Out : INT := 10; (* 20mV = 2 x (10V / 4000 = 0.0025V := 0.003 V := 10 mV) *)
	Tolleranza_OutX: INT := 20; (* 30mV = 10 mV + (10V /  800 = 0.0125V := 0.020 V := 20 mV) *)
	Tolleranza_Tamb_min : INT := 10;
	Tolleranza_RPM : INT := 100;
	Tolleranza_VCC_set : INT := 10; (* 0.01 V *)
	Tolleranza_mA_max : INT := 10; (* 0.01 mA *)
	Tolleranza_VCC_fbk : INT := 100; (* 0.1 V *)
	Tolleranza_mA_fbk : INT := 100; (* 0.1 mA *)
END_VAR

	if TST_DigIn_1  then OK_DigIn_1 := (RES_DigIn_1 = VAL_DigIn_1);  end_if;
	if TST_DigIn_2  then OK_DigIn_2 := (RES_DigIn_2 = VAL_DigIn_2);  end_if;
	if TST_DigIn_3  then OK_DigIn_3 := (RES_DigIn_3 = VAL_DigIn_3);  end_if;
	if TST_DigIn_4  then OK_DigIn_4 := (RES_DigIn_4 = VAL_DigIn_4);  end_if;
	if TST_DigIn_5  then OK_DigIn_5 := (RES_DigIn_5 = VAL_DigIn_5);  end_if;
	if TST_DigIn_6  then OK_DigIn_6 := (RES_DigIn_6 = VAL_DigIn_6);  end_if;
	if TST_DigIn_7  then OK_DigIn_7 := (RES_DigIn_7 = VAL_DigIn_7);  end_if;
	if TST_DigIn_8  then OK_DigIn_8 := (RES_DigIn_8 = VAL_DigIn_8);  end_if;
	if TST_DigIn_9  then OK_DigIn_9 := (RES_DigIn_9 = VAL_DigIn_9);  end_if;
	if TST_DigIn_10 then OK_DigIn_10:= (RES_DigIn_10 = VAL_DigIn_10); end_if;
	if TST_DigIn_11 then OK_DigIn_11:= (RES_DigIn_11 = VAL_DigIn_11); end_if;
	if TST_DigIn_12 then OK_DigIn_12:= (RES_DigIn_12 = VAL_DigIn_12); end_if;
	if TST_DigIn_13 then OK_DigIn_13:= (RES_DigIn_13 = VAL_DigIn_13); end_if;
	if TST_DigIn_14 then OK_DigIn_14:= (RES_DigIn_14 = VAL_DigIn_14); end_if;
	if TST_DigIn_15 then OK_DigIn_15:= (RES_DigIn_15 = VAL_DigIn_15); end_if;
	if TST_DigIn_16 then OK_DigIn_16:= (RES_DigIn_16 = VAL_DigIn_16); end_if;

	if TST_DigOut_1  then OK_DigOut_1 := (RES_DigOut_1 = VAL_DigOut_1);  end_if;
	if TST_DigOut_2  then OK_DigOut_2 := (RES_DigOut_2 = VAL_DigOut_2);  end_if;
	if TST_DigOut_3  then OK_DigOut_3 := (RES_DigOut_3 = VAL_DigOut_3);  end_if;
	if TST_DigOut_4  then OK_DigOut_4 := (RES_DigOut_4 = VAL_DigOut_4);  end_if;
	if TST_DigOut_5  then OK_DigOut_5 := (RES_DigOut_5 = VAL_DigOut_5);  end_if;
	if TST_DigOut_6  then OK_DigOut_6 := (RES_DigOut_6 = VAL_DigOut_6);  end_if;
	if TST_DigOut_7  then OK_DigOut_7 := (RES_DigOut_7 = VAL_DigOut_7);  end_if;
	if TST_DigOut_8  then OK_DigOut_8 := (RES_DigOut_8 = VAL_DigOut_8);  end_if;
	if TST_DigOut_9  then OK_DigOut_9 := (RES_DigOut_9 = VAL_DigOut_9);  end_if;
	if TST_DigOut_10 then OK_DigOut_10:= (RES_DigOut_10 = VAL_DigOut_10); end_if;
	if TST_DigOut_11 then OK_DigOut_11:= (RES_DigOut_11 = VAL_DigOut_11); end_if;
	if TST_DigOut_12 then OK_DigOut_12:= (RES_DigOut_12 = VAL_DigOut_12); end_if;
	if TST_DigOut_13 then OK_DigOut_13:= (RES_DigOut_13 = VAL_DigOut_13); end_if;
	if TST_DigOut_14 then OK_DigOut_14:= (RES_DigOut_14 = VAL_DigOut_14); end_if;
	if TST_DigOut_15 then OK_DigOut_15:= (RES_DigOut_15 = VAL_DigOut_15); end_if;
	if TST_DigOut_16 then OK_DigOut_16:= (RES_DigOut_16 = VAL_DigOut_16); end_if;

	if TST_AnIn_1  then OK_AnIn_1  := abs(RES_AnIn_1  - VAL_AnIn_1 ) <= Tolleranza_In; end_if;
	if TST_AnIn_2  then OK_AnIn_2  := abs(RES_AnIn_2  - VAL_AnIn_2 ) <= Tolleranza_In; end_if;
	if TST_AnIn_3  then OK_AnIn_3  := abs(RES_AnIn_3  - VAL_AnIn_3 ) <= Tolleranza_In; end_if;
	if TST_AnIn_4  then OK_AnIn_4  := abs(RES_AnIn_4  - VAL_AnIn_4 ) <= Tolleranza_In; end_if;

	if TST_AnIn_5  then OK_AnIn_5  := abs(RES_AnIn_5  - VAL_AnIn_5 ) <= Tolleranza_In; end_if;
	if TST_AnIn_6  then OK_AnIn_6  := abs(RES_AnIn_6  - VAL_AnIn_6 ) <= Tolleranza_In; end_if;
	if TST_AnIn_7  then OK_AnIn_7  := abs(RES_AnIn_7  - VAL_AnIn_7 ) <= Tolleranza_In; end_if;
	if TST_AnIn_8  then OK_AnIn_8  := abs(RES_AnIn_8  - VAL_AnIn_8 ) <= Tolleranza_In; end_if;
	if TST_AnIn_9  then OK_AnIn_9  := abs(RES_AnIn_9  - VAL_AnIn_9 ) <= Tolleranza_In; end_if;
	if TST_AnIn_10 then OK_AnIn_10 := abs(RES_AnIn_10 - VAL_AnIn_10) <= Tolleranza_In; end_if;
	if TST_AnIn_11 then OK_AnIn_11 := abs(RES_AnIn_11 - VAL_AnIn_11) <= Tolleranza_In; end_if;
	if TST_AnIn_12 then OK_AnIn_12 := abs(RES_AnIn_12 - VAL_AnIn_12) <= Tolleranza_In; end_if;

	(* input on TPAC1007_4AA 12bit *)
	if TST_AnOut_1  then OK_AnOut_1 := abs(RES_AnOut_1 - VAL_AnOut_1) <= Tolleranza_Out; end_if;
	if TST_AnOut_2  then OK_AnOut_2 := abs(RES_AnOut_2 - VAL_AnOut_2) <= Tolleranza_Out; end_if;
	(* input on TPLC005 10bit *)
	if TST_AnOut_3  then OK_AnOut_3 := abs(RES_AnOut_3 - VAL_AnOut_3) <= Tolleranza_OutX; end_if;
	if TST_AnOut_4  then OK_AnOut_4 := abs(RES_AnOut_4 - VAL_AnOut_4) <= Tolleranza_OutX; end_if;

	if TST_Tamb  then OK_Tamb  := (Tolleranza_Tamb_min <= RES_Tamb) and (RES_Tamb <= VAL_Tamb ); end_if;
	if TST_RPM  then OK_RPM  := abs(UINT_TO_INT(RES_RPM) - UINT_TO_INT(VAL_RPM) ) <= Tolleranza_RPM; end_if;

	if TST_VCC_set  then OK_VCC_set  := abs(RES_VCC_set  - VAL_VCC_set ) <= Tolleranza_VCC_set; end_if;
	if TST_mA_max  then OK_mA_max  := abs(RES_mA_max - VAL_mA_max ) <= Tolleranza_mA_max; end_if;

	if TST_VCC_fbk  then OK_VCC_fbk  := abs(RES_VCC_fbk  - VAL_VCC_fbk ) <= Tolleranza_VCC_fbk; end_if;
	if TST_mA_fbk  then OK_mA_fbk := abs(RES_mA_fbk - VAL_mA_fbk ) <= Tolleranza_mA_fbk; end_if;

	if TST_FWrevision  then OK_FWrevision  := (RES_FWrevision = VAL_FWrevision); end_if;
	if TST_HWconfig  then OK_HWconfig  := (RES_HWconfig = VAL_HWconfig); end_if;

	if TST_RTUS_WR  then OK_RTUS_WR  := (RES_RTUS_WR = VAL_RTUS_WR); end_if;
	if TST_RTUS_RD  then OK_RTUS_RD  := (RES_RTUS_RD = VAL_RTUS_RD); end_if;
	if TST_RTU1_WR  then OK_RTU1_WR  := (RES_RTU1_WR = VAL_RTU1_WR); end_if;
	if TST_RTU1_RD  then OK_RTU1_RD  := (RES_RTU1_RD = VAL_RTU1_RD); end_if;
	if TST_RTU3_WR  then OK_RTU3_WR  := (RES_RTU3_WR = VAL_RTU3_WR); end_if;
	if TST_RTU3_RD  then OK_RTU3_RD  := (RES_RTU3_RD = VAL_RTU3_RD); end_if;
	if TST_CAN1_WR  then OK_CAN1_WR  := (RES_CAN1_WR = VAL_CAN1_WR); end_if;
	if TST_CAN1_RD  then OK_CAN1_RD  := (RES_CAN1_RD = VAL_CAN1_RD); end_if;

END_FUNCTION

(* ---- ClearOK.st ---- *)
(*[[
]]*)
FUNCTION ClearOK
#import "Crosstable.gvl"
VAR_INPUT
END_VAR

	OK_DigIn_1 := FALSE;
	OK_DigIn_2 := FALSE;
	OK_DigIn_3 := FALSE;
	OK_DigIn_4 := FALSE;
	OK_DigIn_5 := FALSE;
	OK_DigIn_6 := FALSE;
	OK_DigIn_7 := FALSE;
	OK_DigIn_8 := FALSE;
	OK_DigIn_9 := FALSE;
	OK_DigIn_10 := FALSE;
	OK_DigIn_11 := FALSE;
	OK_DigIn_12 := FALSE;
	OK_DigIn_13 := FALSE;
	OK_DigIn_14 := FALSE;
	OK_DigIn_15 := FALSE;
	OK_DigIn_16 := FALSE;

	OK_DigOut_1 := FALSE;
	OK_DigOut_2 := FALSE;
	OK_DigOut_3 := FALSE;
	OK_DigOut_4 := FALSE;
	OK_DigOut_5 := FALSE;
	OK_DigOut_6 := FALSE;
	OK_DigOut_7 := FALSE;
	OK_DigOut_8 := FALSE;
	OK_DigOut_9 := FALSE;
	OK_DigOut_10 := FALSE;
	OK_DigOut_11 := FALSE;
	OK_DigOut_12 := FALSE;
	OK_DigOut_13 := FALSE;
	OK_DigOut_14 := FALSE;
	OK_DigOut_15 := FALSE;
	OK_DigOut_16 := FALSE;

	OK_AnIn_1 := FALSE;
	OK_AnIn_2 := FALSE;
	OK_AnIn_3 := FALSE;
	OK_AnIn_4 := FALSE;
	OK_AnIn_5 := FALSE;
	OK_AnIn_6 := FALSE;
	OK_AnIn_7 := FALSE;
	OK_AnIn_8 := FALSE;
	OK_AnIn_9 := FALSE;
	OK_AnIn_10 := FALSE;
	OK_AnIn_11 := FALSE;
	OK_AnIn_12 := FALSE;

	OK_AnOut_1 := FALSE;
	OK_AnOut_2 := FALSE;
	OK_AnOut_3 := FALSE;
	OK_AnOut_4 := FALSE;

	OK_Tamb := FALSE;
	OK_RPM := FALSE;
	OK_VCC_set := FALSE;
	OK_mA_max := FALSE;
	OK_VCC_fbk := FALSE;
	OK_mA_fbk := FALSE;
	OK_FWrevision := FALSE;
	OK_HWconfig := FALSE;

	OK_RTUS_WR := FALSE;
	OK_RTUS_RD := FALSE;
	OK_RTU1_WR := FALSE;
	OK_RTU1_RD := FALSE;
	OK_RTU3_WR := FALSE;
	OK_RTU3_RD := FALSE;
	OK_CAN1_WR := FALSE;
	OK_CAN1_RD := FALSE;

END_FUNCTION

(* ---- ClearPLC.st ---- *)
(*[[
]]*)
FUNCTION ClearPLC
#import "Crosstable.gvl"
VAR_INPUT
END_VAR

	RTU_DigOut_1 := FALSE;
	RTU_DigOut_2 := FALSE;
	RTU_DigOut_3 := FALSE;
	RTU_DigOut_4 := FALSE;
	RTU_DigOut_5 := FALSE;
	RTU_DigOut_6 := FALSE;
	RTU_DigOut_7 := FALSE;
	RTU_DigOut_8 := FALSE;
	RTU_DigOut_9 := FALSE;
	RTU_DigOut_10 := FALSE;
	RTU_DigOut_11 := FALSE;
	RTU_DigOut_12 := FALSE;
	RTU_DigOut_13 := FALSE;
	RTU_DigOut_14 := FALSE;
	RTU_DigOut_15 := FALSE;
	RTU_DigOut_16 := FALSE;

	RTU_AnOut_1 := 0;
	RTU_AnOut_2 := 0;
	RTU_AnOut_3 := 0;
	RTU_AnOut_4 := 0;
	RTU_AnOut_5 := 0;
	RTU_AnOut_6 := 0;
	RTU_AnOut_7 := 0;
	RTU_AnOut_8 := 0;

	PLC_AnOutConf_1 := 2;
	PLC_AnOutConf_2 := 2;
	PLC_AnOut_1 := 0;
	PLC_AnOut_2 := 0;

END_FUNCTION

(* ---- ClearResults.st ---- *)
(*[[
]]*)
FUNCTION ClearResults
#import "Crosstable.gvl"
VAR_INPUT
END_VAR

OK_DigIn_1 := FALSE;
OK_DigIn_2 := FALSE;
OK_DigIn_3 := FALSE;
OK_DigIn_4 := FALSE;
OK_DigIn_5 := FALSE;
OK_DigIn_6 := FALSE;
OK_DigIn_7 := FALSE;
OK_DigIn_8 := FALSE;
OK_DigIn_9 := FALSE;
OK_DigIn_10 := FALSE;
OK_DigIn_11 := FALSE;
OK_DigIn_12 := FALSE;
OK_DigIn_13 := FALSE;
OK_DigIn_14 := FALSE;
OK_DigIn_15 := FALSE;
OK_DigIn_16 := FALSE;
OK_DigOut_1 := FALSE;
OK_DigOut_2 := FALSE;
OK_DigOut_3 := FALSE;
OK_DigOut_4 := FALSE;
OK_DigOut_5 := FALSE;
OK_DigOut_6 := FALSE;
OK_DigOut_7 := FALSE;
OK_DigOut_8 := FALSE;
OK_DigOut_9 := FALSE;
OK_DigOut_10 := FALSE;
OK_DigOut_11 := FALSE;
OK_DigOut_12 := FALSE;
OK_DigOut_13 := FALSE;
OK_DigOut_14 := FALSE;
OK_DigOut_15 := FALSE;
OK_DigOut_16 := FALSE;
OK_AnIn_1 := FALSE;
OK_AnIn_2 := FALSE;
OK_AnIn_3 := FALSE;
OK_AnIn_4 := FALSE;
OK_AnIn_5 := FALSE;
OK_AnIn_6 := FALSE;
OK_AnIn_7 := FALSE;
OK_AnIn_8 := FALSE;
OK_AnIn_9 := FALSE;
OK_AnIn_10 := FALSE;
OK_AnIn_11 := FALSE;
OK_AnIn_12 := FALSE;
OK_AnOut_1 := FALSE;
OK_AnOut_2 := FALSE;
OK_AnOut_3 := FALSE;
OK_AnOut_4 := FALSE;
OK_Tamb := FALSE;
OK_RPM := FALSE;
OK_VCC_set := FALSE;
OK_mA_max := FALSE;
OK_VCC_fbk := FALSE;
OK_mA_fbk := FALSE;
OK_FWrevision := FALSE;
OK_HWconfig := FALSE;
OK_RTUS_WR := FALSE;
OK_RTUS_RD := FALSE;
OK_RTU1_WR := FALSE;
OK_RTU1_RD := FALSE;
OK_RTU3_WR := FALSE;
OK_RTU3_RD := FALSE;
OK_CAN1_WR := FALSE;
OK_CAN1_RD := FALSE;

END_FUNCTION

(* ---- ReadRES.st ---- *)
(*[[
]]*)
FUNCTION ReadRES
#import "Crosstable.gvl"
VAR_INPUT
END_VAR

	if TST_DigIn_1  then RES_DigIn_1 := RESx_DigIn_1;  end_if;
	if TST_DigIn_2  then RES_DigIn_2 := RESx_DigIn_2;  end_if;
	if TST_DigIn_3  then RES_DigIn_3 := RESx_DigIn_3;  end_if;
	if TST_DigIn_4  then RES_DigIn_4 := RESx_DigIn_4;  end_if;
	if TST_DigIn_5  then RES_DigIn_5 := RESx_DigIn_5;  end_if;
	if TST_DigIn_6  then RES_DigIn_6 := RESx_DigIn_6;  end_if;
	if TST_DigIn_7  then RES_DigIn_7 := RESx_DigIn_7;  end_if;
	if TST_DigIn_8  then RES_DigIn_8 := RESx_DigIn_8;  end_if;
	if TST_DigIn_9  then RES_DigIn_9 := RESx_DigIn_9;  end_if;
	if TST_DigIn_10 then RES_DigIn_10:= RESx_DigIn_10; end_if;
	if TST_DigIn_11 then RES_DigIn_11:= RESx_DigIn_11; end_if;
	if TST_DigIn_12 then RES_DigIn_12:= RESx_DigIn_12; end_if;
	if TST_DigIn_13 then RES_DigIn_13:= RESx_DigIn_13; end_if;
	if TST_DigIn_14 then RES_DigIn_14:= RESx_DigIn_14; end_if;
	if TST_DigIn_15 then RES_DigIn_15:= RESx_DigIn_15; end_if;
	if TST_DigIn_16 then RES_DigIn_16:= RESx_DigIn_16; end_if;

	if TST_DigOut_1  then RES_DigOut_1 := RTU_DigIn_1;  end_if;
	if TST_DigOut_2  then RES_DigOut_2 := RTU_DigIn_2;  end_if;
	if TST_DigOut_3  then RES_DigOut_3 := RTU_DigIn_3;  end_if;
	if TST_DigOut_4  then RES_DigOut_4 := RTU_DigIn_4;  end_if;
	if TST_DigOut_5  then RES_DigOut_5 := RTU_DigIn_5;  end_if;
	if TST_DigOut_6  then RES_DigOut_6 := RTU_DigIn_6;  end_if;
	if TST_DigOut_7  then RES_DigOut_7 := RTU_DigIn_7;  end_if;
	if TST_DigOut_8  then RES_DigOut_8 := RTU_DigIn_8;  end_if;
	if TST_DigOut_9  then RES_DigOut_9 := RTU_DigIn_9;  end_if;
	if TST_DigOut_10 then RES_DigOut_10:= RTU_DigIn_10; end_if;
	if TST_DigOut_11 then RES_DigOut_11:= RTU_DigIn_11; end_if;
	if TST_DigOut_12 then RES_DigOut_12:= RTU_DigIn_12; end_if;
	if TST_DigOut_13 then RES_DigOut_13:= RTU_DigIn_13; end_if;
	if TST_DigOut_14 then RES_DigOut_14:= RTU_DigIn_14; end_if;
	if TST_DigOut_15 then RES_DigOut_15:= RTU_DigIn_15; end_if;
	if TST_DigOut_16 then RES_DigOut_16:= RTU_DigIn_16; end_if;

	if TST_AnIn_1  then RES_AnIn_1  := RESx_AnIn_1;  end_if;
	if TST_AnIn_2  then RES_AnIn_2  := RESx_AnIn_2;  end_if;
	if TST_AnIn_3  then RES_AnIn_3  := RESx_AnIn_3;  end_if;
	if TST_AnIn_4  then RES_AnIn_4  := RESx_AnIn_4;  end_if;

	if TST_AnIn_5  then RES_AnIn_5  := RESx_AnIn_5;  end_if;
	if TST_AnIn_6  then RES_AnIn_6  := RESx_AnIn_6;  end_if;
	if TST_AnIn_7  then RES_AnIn_7  := RESx_AnIn_7;  end_if;
	if TST_AnIn_8  then RES_AnIn_8  := RESx_AnIn_8;  end_if;
	if TST_AnIn_9  then RES_AnIn_9  := RESx_AnIn_9;  end_if;
	if TST_AnIn_10 then RES_AnIn_10 := RESx_AnIn_10;  end_if;
	if TST_AnIn_11 then RES_AnIn_11 := RESx_AnIn_11;  end_if;
	if TST_AnIn_12 then RES_AnIn_12 := RESx_AnIn_12;  end_if;

	if TST_AnOut_1  then RES_AnOut_1 := RES2_AnIn_1 / 10;  end_if;
	if TST_AnOut_2  then RES_AnOut_2 := RES2_AnIn_2 / 10;  end_if;
	if TST_AnOut_3  then RES_AnOut_3 := RTU_AnIn_1 / 10;  end_if;
	if TST_AnOut_4  then RES_AnOut_4 := RTU_AnIn_2 / 10;  end_if;

	if TST_Tamb  then RES_Tamb  := RESx_Tamb;  end_if;
	if TST_RPM   then RES_RPM  := RESx_RPM;  end_if;

	if TST_VCC_set  then RES_VCC_set  := PLC_AnOut_3;  end_if;
	if TST_mA_max  then RES_mA_max  := PLC_AnOut_4;  end_if;

	if TST_VCC_fbk  then RES_VCC_fbk  := PLC_AnIn_1;  end_if;
	if TST_mA_fbk  then RES_mA_fbk  := PLC_AnIn_2;  end_if;

	if TST_FWrevision  then RES_FWrevision  := RESx_FWrevision;  end_if;
	if TST_HWconfig  then RES_HWconfig  := RESx_HWconfig;  end_if;

	if TST_RTU1_WR then RES_RTU1_WR := RES2_RTUS_RD; end_if;
	if TST_RTU1_RD then RES_RTU1_RD := RESx_RTU1_RD; end_if;
	if TST_RTU3_RD then RES_RTU3_RD := RESx_RTU3_RD; end_if;

	if TST_CAN1_WR then RES_CAN1_WR := RESx_CAN1_RD; end_if;
	if TST_CAN1_RD then RES_CAN1_RD := RESx_CAN1_RD; end_if;

END_FUNCTION

(* ---- Translate_AnIn.st ---- *)
(*[[
]]*)
FUNCTION Translate_AnIn
#import "Crosstable.gvl"
VAR_INPUT
END_VAR

	if TST_AnIn_1  then
		TSTx_AnIn_1 := TRUE;
		VALx_AnInConf_1 := VAL_AnInConf_1;
		VALx_AnInFltr_1 := VAL_AnInFltr_1;
		(* <-- Head AO1 + DO6 + DO8 *)
		PLC_AnOutConf_1 := VAL_AnInConf_1;
		PLC_AnOut_1 := VAL_AnIn_1;
		PLC_DigDir_6 := 1;
		PLC_DigDir_8 := 1;
		case VAL_AnInConf_1 of
		1: PLC_DigOut_8 := 1; PLC_DigOut_6 := 0;
		2: PLC_DigOut_8 := 0; PLC_DigOut_6 := 0;
		3, 4, 5, 6, 7: PLC_DigOut_8 := 0; PLC_DigOut_6 := 1;
		else PLC_DigOut_8 := 0; PLC_DigOut_6 := 0;
		end_case;
	end_if;

	if TST_AnIn_2  then
		TSTx_AnIn_2 := TRUE;
		VALx_AnInConf_2 := VAL_AnInConf_2;
		VALx_AnInFltr_2 := VAL_AnInFltr_2;
		(* <-- Head AO2 + DO5 + DO7 *)
		PLC_AnOutConf_2 := VAL_AnInConf_2;
		PLC_AnOut_2 := VAL_AnIn_2;
		PLC_DigDir_5 := 1;
		PLC_DigDir_7 := 1;
		case VAL_AnInConf_2 of
		1: PLC_DigOut_7 := 1; PLC_DigOut_5 := 0;
		2: PLC_DigOut_7 := 0; PLC_DigOut_5 := 0;
		3, 4, 5, 6, 7: PLC_DigOut_7 := 0; PLC_DigOut_5 := 1;
		else PLC_DigOut_7 := 0; PLC_DigOut_5 := 0;
		end_case;
	end_if;

	if TST_AnIn_3  then
		TSTx_AnIn_3 := TRUE;
		VALx_AnInConf_3 := VAL_AnInConf_3;
		VALx_AnInFltr_3 := VAL_AnInFltr_3;
		(* <-- Horn2 AO1 + DO6 + DO8 *)
		TST2_AnOut_1 := 1;
		VAL2_AnOutConf_1 := VAL_AnInConf_3;
		VAL2_AnOut_1 := VAL_AnIn_3;
		TST2_DigOut_6 := 1;
		TST2_DigOut_8 := 1;
		case VAL_AnInConf_3 of
		1: VAL2_DigOut_8 := 1; VAL2_DigOut_6 := 0;
		2: VAL2_DigOut_8 := 0; VAL2_DigOut_6 := 0;
		3, 4, 5, 6, 7: VAL2_DigOut_8 := 0; VAL2_DigOut_6 := 1;
		else VAL2_DigOut_8 := 0; VAL2_DigOut_6 := 0;
		end_case;
	end_if;

	if TST_AnIn_4  then
		TSTx_AnIn_4 := TRUE;
		VALx_AnInConf_4 := VAL_AnInConf_4;
		VALx_AnInFltr_4 := VAL_AnInFltr_4;
		(* <-- Horn2 AO2 + DO5 + DO7 *)
		TST2_AnOut_2 := 1;
		VAL2_AnOutConf_2 := VAL_AnInConf_4;
		VAL2_AnOut_3 := VAL_AnIn_4;
		TST2_DigOut_5 := 1;
		TST2_DigOut_7 := 1;
		case VAL_AnInConf_4 of
		1: VAL2_DigOut_7 := 1; VAL2_DigOut_5 := 0;
		2: VAL2_DigOut_7 := 0; VAL2_DigOut_5 := 0;
		3, 4, 5, 6, 7: VAL2_DigOut_7 := 0; VAL2_DigOut_5 := 1;
		else VAL2_DigOut_7 := 0; VAL2_DigOut_5 := 0;
		end_case;
	end_if;

	if TST_AnIn_5  then
		TSTx_AnIn_5 := TRUE;
		VALx_AnInConf_5 := VAL_AnInConf_5;
		VALx_AnInFltr_5 := VAL_AnInFltr_5;
		(* <-- Head/TPLC005 AO1 *)
		RTU_AnOut_1 := VAL_AnIn_5;
		(* <-- Horn2 AO4 V : double for TPAC1007_4AB *)
		TST2_AnOut_4 := 1;
		VAL2_AnOutConf_4 := VAL_AnInConf_5;
		VAL2_AnOut_4 := VAL_AnIn_5;
	end_if;
	if TST_AnIn_6  then
		TSTx_AnIn_6 := TRUE;
		VALx_AnInConf_6 := VAL_AnInConf_6;
		VALx_AnInFltr_6 := VAL_AnInFltr_6;
		(* <-- Head/TPLC005 AO2 *)
		RTU_AnOut_2 := VAL_AnIn_6;
	end_if;
	if TST_AnIn_7  then
		TSTx_AnIn_7 := TRUE;
		VALx_AnInConf_7 := VAL_AnInConf_7;
		VALx_AnInFltr_7 := VAL_AnInFltr_7;
		(* <-- Head/TPLC005 AO3 *)
		PLC_AnOut_3 := VAL_AnIn_7;
	end_if;
	if TST_AnIn_8  then
		TSTx_AnIn_8 := TRUE;
		VALx_AnInConf_8 := VAL_AnInConf_8;
		VALx_AnInFltr_8 := VAL_AnInFltr_8;
		(* <-- Head/TPLC005 AO4 *)
		RTU_AnOut_4 := VAL_AnIn_8;
	end_if;
	if TST_AnIn_9  then
		TSTx_AnIn_9 := TRUE;
		VALx_AnInConf_9 := VAL_AnInConf_9;
		VALx_AnInFltr_9 := VAL_AnInFltr_9;
		(* <-- Head/TPLC005 AO5*)
		RTU_AnOut_5 := VAL_AnIn_9;
	end_if;
	if TST_AnIn_10 then
		TSTx_AnIn_10:= TRUE;
		VALx_AnInConf_10:= VAL_AnInConf_10;
		VALx_AnInFltr_10:= VAL_AnInFltr_10;
		(* <-- Head/TPLC005 AO6*)
		RTU_AnOut_6 := VAL_AnIn_10;
	end_if;
	if TST_AnIn_11 then
		TSTx_AnIn_11:= TRUE;
		VALx_AnInConf_11:= VAL_AnInConf_11;
		VALx_AnInFltr_11:= VAL_AnInFltr_11;
		(* <-- Head/TPLC005 AO7*)
		RTU_AnOut_7 := VAL_AnIn_11;
	end_if;
	if TST_AnIn_12 then
		TSTx_AnIn_12:= TRUE;
		VALx_AnInConf_12:= VAL_AnInConf_12;
		VALx_AnInFltr_12:= VAL_AnInFltr_12;
		(* <-- Head/TPLC005 AO8*)
		RTU_AnOut_8 := VAL_AnIn_12;
	end_if;

END_FUNCTION

(* ---- Translate_AnOut.st ---- *)
(*[[
]]*)
FUNCTION Translate_AnOut
#import "Crosstable.gvl"
VAR_INPUT
END_VAR

	if TST_AnOut_1  then
		TSTx_AnOut_1 := TRUE;
		VALx_AnOut_1 := VAL_AnOut_1;
		VALx_AnOutConf_1 := VAL_AnOutConf_1;
		(* --> Horn2 AI1 + DO4 *)
		TST2_AnIn_1 := 1;
		VAL2_AnInConf_1 := VAL_AnOutConf_1;
		VAL2_AnInFltr_1 := 16;
		TST2_DigOut_4 := 1;
		case VAL_AnOutConf_1 of
		1: VAL2_DigOut_4 := 1;
		2: VAL2_DigOut_4 := 0;
		end_case;
	end_if;

	if TST_AnOut_2  then
		TSTx_AnOut_2 := TRUE;
		VALx_AnOut_2 := VAL_AnOut_2;
		VALx_AnOutConf_2 := VAL_AnOutConf_2;
		(* --> Horn2 AI2 + DO3 *)
		TST2_AnIn_2 := 1;
		VAL2_AnInConf_2 := VAL_AnOutConf_2;
		VAL2_AnInFltr_2 := 16;
		TST2_DigOut_3 := 1;
		case VAL_AnOutConf_2 of
		1: VAL2_DigOut_3 := 1;
		2: VAL2_DigOut_3 := 0;
		end_case;
	end_if;

	if TST_AnOut_3  then
		TSTx_AnOut_3 := TRUE;
		VALx_AnOut_3 := VAL_AnOut_3;
		VALx_AnOutConf_3 := VAL_AnOutConf_3;
		(* --> Head/TPLC005 AI1 *)
		PLC_AnInConf_1 := VAL_AnOutConf_3;
	end_if;

	if TST_AnOut_4  then
		TSTx_AnOut_4 := TRUE;
		VALx_AnOut_4 := VAL_AnOut_4;
		VALx_AnOutConf_4 := VAL_AnOutConf_4;
		(* --> Head/TPLC005 AI2 *)
		PLC_AnInConf_2 := VAL_AnOutConf_4;
	end_if;

END_FUNCTION

(* ---- Translate_DigIn.st ---- *)
(*[[
]]*)
FUNCTION Translate_DigIn
#import "Crosstable.gvl"
VAR_INPUT
END_VAR

	(* DigIn 1..16 are on the local TPLC005 *)
	TSTx_DigIn_1 := TST_DigIn_1;
	TSTx_DigIn_2 := TST_DigIn_2;
	TSTx_DigIn_3 := TST_DigIn_3;
	TSTx_DigIn_4 := TST_DigIn_4;
	TSTx_DigIn_5 := TST_DigIn_5;
	TSTx_DigIn_6 := TST_DigIn_6;
	TSTx_DigIn_7 := TST_DigIn_7;
	TSTx_DigIn_8 := TST_DigIn_8;
	TSTx_DigIn_9 := TST_DigIn_9;
	TSTx_DigIn_10:= TST_DigIn_10;
	TSTx_DigIn_11:= TST_DigIn_11;
	TSTx_DigIn_12:= TST_DigIn_12;
	TSTx_DigIn_13:= TST_DigIn_13;
	TSTx_DigIn_14:= TST_DigIn_14;
	TSTx_DigIn_15:= TST_DigIn_15;
	TSTx_DigIn_16:= TST_DigIn_16;

	if TST_DigIn_1  then RTU_DigOut_1 := VAL_DigIn_1;  end_if;
	if TST_DigIn_2  then RTU_DigOut_2 := VAL_DigIn_2;  end_if;
	if TST_DigIn_3  then RTU_DigOut_3 := VAL_DigIn_3;  end_if;
	if TST_DigIn_4  then RTU_DigOut_4 := VAL_DigIn_4;  end_if;
	if TST_DigIn_5  then RTU_DigOut_5 := VAL_DigIn_5;  end_if;
	if TST_DigIn_6  then RTU_DigOut_6 := VAL_DigIn_6;  end_if;
	if TST_DigIn_7  then RTU_DigOut_7 := VAL_DigIn_7;  end_if;
	if TST_DigIn_8  then RTU_DigOut_8 := VAL_DigIn_8;  end_if;
	if TST_DigIn_9  then RTU_DigOut_9 := VAL_DigIn_9;  end_if;
	if TST_DigIn_10 then RTU_DigOut_10:= VAL_DigIn_10; end_if;
	if TST_DigIn_11 then RTU_DigOut_11:= VAL_DigIn_11; end_if;
	if TST_DigIn_12 then RTU_DigOut_12:= VAL_DigIn_12; end_if;
	if TST_DigIn_13 then RTU_DigOut_13:= VAL_DigIn_13; end_if;
	if TST_DigIn_14 then RTU_DigOut_14:= VAL_DigIn_14; end_if;
	if TST_DigIn_15 then RTU_DigOut_15:= VAL_DigIn_15; end_if;
	if TST_DigIn_16 then RTU_DigOut_16:= VAL_DigIn_16; end_if;

END_FUNCTION

(* ---- Translate_DigOut.st ---- *)
(*[[
]]*)
FUNCTION Translate_DigOut
#import "Crosstable.gvl"
VAR_INPUT
END_VAR

	(* DigOut 1..16 are on the local TPLC005 *)
	TSTx_DigOut_1 := TST_DigOut_1;
	TSTx_DigOut_2 := TST_DigOut_2;
	TSTx_DigOut_3 := TST_DigOut_3;
	TSTx_DigOut_4 := TST_DigOut_4;
	TSTx_DigOut_5 := TST_DigOut_5;
	TSTx_DigOut_6 := TST_DigOut_6;
	TSTx_DigOut_7 := TST_DigOut_7;
	TSTx_DigOut_8 := TST_DigOut_8;
	TSTx_DigOut_9 := TST_DigOut_9;
	TSTx_DigOut_10:= TST_DigOut_10;
	TSTx_DigOut_11:= TST_DigOut_11;
	TSTx_DigOut_12:= TST_DigOut_12;
	TSTx_DigOut_13:= TST_DigOut_13;
	TSTx_DigOut_14:= TST_DigOut_14;
	TSTx_DigOut_15:= TST_DigOut_15;
	TSTx_DigOut_16:= TST_DigOut_16;

	if TST_DigOut_1  then VALx_DigOut_1 := VAL_DigOut_1;  end_if;
	if TST_DigOut_2  then VALx_DigOut_2 := VAL_DigOut_2;  end_if;
	if TST_DigOut_3  then VALx_DigOut_3 := VAL_DigOut_3;  end_if;
	if TST_DigOut_4  then VALx_DigOut_4 := VAL_DigOut_4;  end_if;
	if TST_DigOut_5  then VALx_DigOut_5 := VAL_DigOut_5;  end_if;
	if TST_DigOut_6  then VALx_DigOut_6 := VAL_DigOut_6;  end_if;
	if TST_DigOut_7  then VALx_DigOut_7 := VAL_DigOut_7;  end_if;
	if TST_DigOut_8  then VALx_DigOut_8 := VAL_DigOut_8;  end_if;
	if TST_DigOut_9  then VALx_DigOut_9 := VAL_DigOut_9;  end_if;
	if TST_DigOut_10 then VALx_DigOut_10:= VAL_DigOut_10; end_if;
	if TST_DigOut_11 then VALx_DigOut_11:= VAL_DigOut_11; end_if;
	if TST_DigOut_12 then VALx_DigOut_12:= VAL_DigOut_12; end_if;
	if TST_DigOut_13 then VALx_DigOut_13:= VAL_DigOut_13; end_if;
	if TST_DigOut_14 then VALx_DigOut_14:= VAL_DigOut_14; end_if;
	if TST_DigOut_15 then VALx_DigOut_15:= VAL_DigOut_15; end_if;
	if TST_DigOut_16 then VALx_DigOut_16:= VAL_DigOut_16; end_if;

END_FUNCTION

(* ---- Translate_Others.st ---- *)
(*[[
]]*)
FUNCTION Translate_Others
#import "Crosstable.gvl"
VAR_INPUT
END_VAR

	if TST_Tamb  then
		TSTx_Tamb := TRUE;
	end_if;

	if TST_RPM  then
		TSTx_RPM := TRUE;
		(* <-- Horn2 AO3 PWM *)
		TST2_AnOut_3 := 1;
		VAL2_AnOutConf_3 := 3; (* PWM *)
		VAL2_AnOut_3 := UINT_TO_INT(VAL_RPM); (* FIXME: conversion ? *)
	end_if;

	if TST_FWrevision  then
		TSTx_FWrevision := TRUE;
	end_if;

	if TST_HWconfig then
		TSTx_HWconfig := TRUE;
	end_if;

	(* only from the testing equipment *)
	if TST_VCC_set then
		(* --> Head AO3 V *)
		PLC_AnOutConf_3 := 2; (* 0..10 V *)
		PLC_AnOut_3 := VAL_VCC_set; (* FIXME: conversion ? *)
	end_if;

	if TST_mA_max then
		(* --> Head AO4 V *)
		PLC_AnOutConf_4 := 2; (* 0..10 V *)
		PLC_AnOut_4 := VAL_mA_max; (* FIXME: conversion ? *)
	end_if;

	if TST_VCC_fbk then
		(* --> Head AI1 V *)
		PLC_AnInConf_1 := 2; (* 0..10 V *)
	end_if;

	if TST_mA_fbk then
		(* --> Head AI2 V *)
		PLC_AnInConf_2 := 2; (* 0..10 V *)
	end_if;

END_FUNCTION

(* ---- WriteTST.st ---- *)
(*[[
]]*)
FUNCTION WriteTST
#import "Crosstable.gvl"
VAR_INPUT
END_VAR

	(* we test the DigIn 1..16 by the TPLC005 16DO module *)
 	TSTx_DigIn_1 := TST_DigIn_1;
	TSTx_DigIn_2 := TST_DigIn_2;
	TSTx_DigIn_3 := TST_DigIn_3;
	TSTx_DigIn_4 := TST_DigIn_4;
	TSTx_DigIn_5 := TST_DigIn_5;
	TSTx_DigIn_6 := TST_DigIn_6;
	TSTx_DigIn_7 := TST_DigIn_7;
	TSTx_DigIn_8 := TST_DigIn_8;
	TSTx_DigIn_9 := TST_DigIn_9;
	TSTx_DigIn_10:= TST_DigIn_10;
	TSTx_DigIn_11:= TST_DigIn_11;
	TSTx_DigIn_12:= TST_DigIn_12;
	TSTx_DigIn_13:= TST_DigIn_13;
	TSTx_DigIn_14:= TST_DigIn_14;
	TSTx_DigIn_15:= TST_DigIn_15;
	TSTx_DigIn_16:= TST_DigIn_16;
    (* no TST2_DigIn_* *)

    (* we test the DigOut 1..16 by the TPLC005 16DI module *)
	TSTx_DigOut_1 := TST_DigOut_1;
	TSTx_DigOut_2 := TST_DigOut_2;
	TSTx_DigOut_3 := TST_DigOut_3;
	TSTx_DigOut_4 := TST_DigOut_4;
	TSTx_DigOut_5 := TST_DigOut_5;
	TSTx_DigOut_6 := TST_DigOut_6;
	TSTx_DigOut_7 := TST_DigOut_7;
	TSTx_DigOut_8 := TST_DigOut_8;
	TSTx_DigOut_9 := TST_DigOut_9;
	TSTx_DigOut_10:= TST_DigOut_10;
	TSTx_DigOut_11:= TST_DigOut_11;
	TSTx_DigOut_12:= TST_DigOut_12;
	TSTx_DigOut_13:= TST_DigOut_13;
	TSTx_DigOut_14:= TST_DigOut_14;
	TSTx_DigOut_15:= TST_DigOut_15;
	TSTx_DigOut_16:= TST_DigOut_16;
    (* no TST2_DigOut_* *)

    (* we test the AnIn 1..2 by the local AnOut 1..2 and local DigOut 5..8 *)
	TSTx_AnIn_1 := TST_AnIn_1;
	TSTx_AnIn_2 := TST_AnIn_2;

    (* we test the AnIn 3..4 by the Horn TPAC1007_4AA AnOut 1..2 and local DigOut 5..8 *)
	TSTx_AnIn_3 := TST_AnIn_3;
    TST2_AnOut_1 := TST_AnIn_3;
    TST2_DigOut_6 := TRUE;
    TST2_DigOut_8 := TRUE;

	TSTx_AnIn_4 := TST_AnIn_4;
    TST2_AnOut_2 := TST_AnIn_4;
    TST2_DigOut_5 := TRUE;
    TST2_DigOut_7 := TRUE;

    (* we test the AnIn 5..12 (PT100 only) by the TPLC005 8AO module (actually internal 8DO) *)
    TST2_AnOut_4:= TST_AnIn_5; (* only TPAC1007_AB *)
	TSTx_AnIn_5 := TST_AnIn_5;
	TSTx_AnIn_6 := TST_AnIn_6;
	TSTx_AnIn_7 := TST_AnIn_7;
	TSTx_AnIn_8 := TST_AnIn_8;
	TSTx_AnIn_9 := TST_AnIn_9;
	TSTx_AnIn_10:= TST_AnIn_10;
	TSTx_AnIn_11:= TST_AnIn_11;
	TSTx_AnIn_12:= TST_AnIn_12;

    (* we test the AnOut 1..2 by both the local AnIn 1..2 and the Horn TPAC1007_4AA AnIn 1..2 and local DigOut 3..4 *)
    TSTx_AnOut_1 := TST_AnOut_1;
    TST2_AnIn_1 := TST_AnOut_1;
    TST2_DigOut_3 := TRUE;

    TSTx_AnOut_2 := TST_AnOut_2;
    TST2_AnIn_2 := TST_AnOut_2;
    TST2_DigOut_4 := TRUE;

    (* we test the AnOut 3..4 by the by the TPLC005 internal 2AI *)
    TSTx_AnOut_3 := TST_AnOut_3;
    TSTx_AnOut_4 := TST_AnOut_4;

    (* we test the Others I/O ...  *)
    TSTx_Tamb := TST_Tamb;
    TSTx_RPM := TST_RPM;
    TSTx_FWrevision := TST_FWrevision;
    TSTx_HWconfig := TST_HWconfig;
    TST2_AnOut_3 := TST_RPM;

	(* RTUS: Head.RTU1 --> Prey.RTUS *)
    TSTx_RTUS_WR := TST_RTUS_WR;
    TSTx_RTUS_RD := TST_RTUS_RD;

	(* RTU1: Prey.RTU1 --> Horn.RTUS *)
    TSTx_RTU1_WR := TST_RTU1_WR;
	TST2_RTUS_RD := TST_RTU1_WR;

    TSTx_RTU1_RD := TST_RTU1_RD;
	TST2_RTUS_WR := TST_RTU1_RD;

	(* RTU3: Prey.RTU3 <--> TPLC005 *)
	TSTx_RTU3_WR := TST_RTU3_WR;
	TSTx_RTU3_RD := TST_RTU3_RD;

	(* CAN1: Prey.CAN1 <--> MPNC010 *)
    TSTx_CAN1_WR := TST_CAN1_WR;
    TSTx_CAN1_RD := TST_CAN1_RD;

END_FUNCTION

(* ---- WriteVAL.st ---- *)
(*[[
]]*)
FUNCTION WriteVAL
#import "Crosstable.gvl"
VAR_INPUT
END_VAR

	if TST_DigIn_1  then RTU_DigOut_1 := VAL_DigIn_1;  end_if;
	if TST_DigIn_2  then RTU_DigOut_2 := VAL_DigIn_2;  end_if;
	if TST_DigIn_3  then RTU_DigOut_3 := VAL_DigIn_3;  end_if;
	if TST_DigIn_4  then RTU_DigOut_4 := VAL_DigIn_4;  end_if;
	if TST_DigIn_5  then RTU_DigOut_5 := VAL_DigIn_5;  end_if;
	if TST_DigIn_6  then RTU_DigOut_6 := VAL_DigIn_6;  end_if;
	if TST_DigIn_7  then RTU_DigOut_7 := VAL_DigIn_7;  end_if;
	if TST_DigIn_8  then RTU_DigOut_8 := VAL_DigIn_8;  end_if;
	if TST_DigIn_9  then RTU_DigOut_9 := VAL_DigIn_9;  end_if;
	if TST_DigIn_10 then RTU_DigOut_10:= VAL_DigIn_10; end_if;
	if TST_DigIn_11 then RTU_DigOut_11:= VAL_DigIn_11; end_if;
	if TST_DigIn_12 then RTU_DigOut_12:= VAL_DigIn_12; end_if;
	if TST_DigIn_13 then RTU_DigOut_13:= VAL_DigIn_13; end_if;
	if TST_DigIn_14 then RTU_DigOut_14:= VAL_DigIn_14; end_if;
	if TST_DigIn_15 then RTU_DigOut_15:= VAL_DigIn_15; end_if;
	if TST_DigIn_16 then RTU_DigOut_16:= VAL_DigIn_16; end_if;

	if TST_DigOut_1  then VALx_DigOut_1 := VAL_DigOut_1;  end_if;
	if TST_DigOut_2  then VALx_DigOut_2 := VAL_DigOut_2;  end_if;
	if TST_DigOut_3  then VALx_DigOut_3 := VAL_DigOut_3;  end_if;
	if TST_DigOut_4  then VALx_DigOut_4 := VAL_DigOut_4;  end_if;
	if TST_DigOut_5  then VALx_DigOut_5 := VAL_DigOut_5;  end_if;
	if TST_DigOut_6  then VALx_DigOut_6 := VAL_DigOut_6;  end_if;
	if TST_DigOut_7  then VALx_DigOut_7 := VAL_DigOut_7;  end_if;
	if TST_DigOut_8  then VALx_DigOut_8 := VAL_DigOut_8;  end_if;
	if TST_DigOut_9  then VALx_DigOut_9 := VAL_DigOut_9;  end_if;
	if TST_DigOut_10 then VALx_DigOut_10:= VAL_DigOut_10; end_if;
	if TST_DigOut_11 then VALx_DigOut_11:= VAL_DigOut_11; end_if;
	if TST_DigOut_12 then VALx_DigOut_12:= VAL_DigOut_12; end_if;
	if TST_DigOut_13 then VALx_DigOut_13:= VAL_DigOut_13; end_if;
	if TST_DigOut_14 then VALx_DigOut_14:= VAL_DigOut_14; end_if;
	if TST_DigOut_15 then VALx_DigOut_15:= VAL_DigOut_15; end_if;
	if TST_DigOut_16 then VALx_DigOut_16:= VAL_DigOut_16; end_if;

	if TST_AnIn_1  then
		VALx_AnInConf_1 := VAL_AnInConf_1;
		VALx_AnInFltr_1 := VAL_AnInFltr_1;
		(* <-- Head AO1 + DO6 + DO8 *)
		PLC_DigDir_6 := 1;
		PLC_DigDir_8 := 1;
		case VAL_AnInConf_1 of
		1: PLC_DigOut_8 := 1; PLC_DigOut_6 := 0; PLC_AnOutConf_1 := VAL_AnInConf_1; PLC_AnOut_1 := VAL_AnIn_1 / 10;
		2: PLC_DigOut_8 := 0; PLC_DigOut_6 := 0; PLC_AnOutConf_1 := VAL_AnInConf_1; PLC_AnOut_1 := VAL_AnIn_1 / 10;
		3, 4, 5, 6: PLC_DigOut_8 := 0; PLC_DigOut_6 := 1; PLC_AnOutConf_1 := VAL_AnInConf_1; PLC_AnOut_1 := VAL_AnIn_1 / 10;
		7: PLC_DigOut_8 := 0; PLC_DigOut_6 := 1;  VAL_AnOut_1 := 0; VAL_AnOutConf_1 := 2;
		else PLC_DigOut_8 := 0; PLC_DigOut_6 := 0;
		end_case;
	end_if;

	if TST_AnIn_2  then
		VALx_AnInConf_2 := VAL_AnInConf_2;
		VALx_AnInFltr_2 := VAL_AnInFltr_2;
		(* <-- Head AO2 + DO5 + DO7 *)
		PLC_DigDir_5 := 1;
		PLC_DigDir_7 := 1;
		case VAL_AnInConf_2 of
		1: PLC_DigOut_7 := 1; PLC_DigOut_5 := 0; PLC_AnOutConf_2 := VAL_AnInConf_2; PLC_AnOut_2 := VAL_AnIn_2 / 10;
		2: PLC_DigOut_7 := 0; PLC_DigOut_5 := 0; PLC_AnOutConf_2 := VAL_AnInConf_2; PLC_AnOut_2 := VAL_AnIn_2 / 10;
		3, 4, 5, 6: PLC_DigOut_7 := 0; PLC_DigOut_5 := 1; PLC_AnOutConf_2 := VAL_AnInConf_2; PLC_AnOut_2 := VAL_AnIn_2 / 10;
		7: PLC_DigOut_8 := 0; PLC_DigOut_6 := 1;  VAL_AnOut_2 := 0; VAL_AnOutConf_2 := 2;
		else PLC_DigOut_7 := 0; PLC_DigOut_5 := 0;
		end_case;
	end_if;

	if TST_AnIn_3  then
		VALx_AnInConf_3 := VAL_AnInConf_3;
		VALx_AnInFltr_3 := VAL_AnInFltr_3;
		(* <-- Horn2 AO1 + DO6 + DO8 *)
		case VAL_AnInConf_3 of
		1: VAL2_DigOut_8 := 1; VAL2_DigOut_6 := 0; VAL2_AnOutConf_1 := VAL_AnInConf_3; VAL2_AnOut_1 := VAL_AnIn_3 / 10;
		2: VAL2_DigOut_8 := 0; VAL2_DigOut_6 := 0; VAL2_AnOutConf_1 := VAL_AnInConf_3; VAL2_AnOut_1 := VAL_AnIn_3 / 10;
		3, 4, 5, 6: VAL2_DigOut_8 := 0; VAL2_DigOut_6 := 1; VAL2_AnOutConf_1 := VAL_AnInConf_3; VAL2_AnOut_1 := VAL_AnIn_3 / 10;
		7: PLC_DigOut_8 := 0; PLC_DigOut_6 := 1;  VAL2_AnOut_3 := 0; VAL2_AnOutConf_3 := 2;
		else VAL2_DigOut_8 := 0; VAL2_DigOut_6 := 0;
		end_case;
	end_if;

	if TST_AnIn_4  then
		VALx_AnInConf_4 := VAL_AnInConf_4;
		VALx_AnInFltr_4 := VAL_AnInFltr_4;
		(* <-- Horn2 AO2 + DO5 + DO7 *)
		case VAL_AnInConf_4 of
		1: VAL2_DigOut_7 := 1; VAL2_DigOut_5 := 0; VAL2_AnOutConf_2 := VAL_AnInConf_4; VAL2_AnOut_2 := VAL_AnIn_4 / 10;
		2: VAL2_DigOut_7 := 0; VAL2_DigOut_5 := 0; VAL2_AnOutConf_2 := VAL_AnInConf_4; VAL2_AnOut_2 := VAL_AnIn_4 / 10;
		3, 4, 5, 6: VAL2_DigOut_7 := 0; VAL2_DigOut_5 := 1; VAL2_AnOutConf_2 := VAL_AnInConf_4; VAL2_AnOut_2 := VAL_AnIn_4 / 10;
		7: PLC_DigOut_8 := 0; PLC_DigOut_6 := 1;  VAL2_AnOut_4 := 0; VAL2_AnOutConf_4 := 2;
		else VAL2_DigOut_7 := 0; VAL2_DigOut_5 := 0;
		end_case;
	end_if;

	if TST_AnIn_5  then
		VALx_AnInConf_5 := VAL_AnInConf_5;
		VALx_AnInFltr_5 := VAL_AnInFltr_5;
		(* <-- Head/TPLC005 AO1 *)
		RTU_AnOut_1 := VAL_AnIn_5 / 10;
		(* <-- Horn2 AO4 V : double for TPAC1007_4AB *)
		VAL2_AnOutConf_4 := VAL_AnInConf_5;
		VAL2_AnOut_4 := VAL_AnIn_5 / 10;
	end_if;
	if TST_AnIn_6  then
		VALx_AnInConf_6 := VAL_AnInConf_6;
		VALx_AnInFltr_6 := VAL_AnInFltr_6;
		(* <-- Head/TPLC005 AO2 *)
		RTU_AnOut_2 := VAL_AnIn_6 / 10;
	end_if;
	if TST_AnIn_7  then
		VALx_AnInConf_7 := VAL_AnInConf_7;
		VALx_AnInFltr_7 := VAL_AnInFltr_7;
		(* <-- Head/TPLC005 AO3 *)
		PLC_AnOut_3 := VAL_AnIn_7 / 10;
	end_if;
	if TST_AnIn_8  then
		VALx_AnInConf_8 := VAL_AnInConf_8;
		VALx_AnInFltr_8 := VAL_AnInFltr_8;
		(* <-- Head/TPLC005 AO4 *)
		RTU_AnOut_4 := VAL_AnIn_8 / 10;
	end_if;
	if TST_AnIn_9  then
		VALx_AnInConf_9 := VAL_AnInConf_9;
		VALx_AnInFltr_9 := VAL_AnInFltr_9;
		(* <-- Head/TPLC005 AO5*)
		RTU_AnOut_5 := VAL_AnIn_9 / 10;
	end_if;
	if TST_AnIn_10 then
		VALx_AnInConf_10:= VAL_AnInConf_10;
		VALx_AnInFltr_10:= VAL_AnInFltr_10;
		(* <-- Head/TPLC005 AO6*)
		RTU_AnOut_6 := VAL_AnIn_10 / 10;
	end_if;
	if TST_AnIn_11 then
		VALx_AnInConf_11:= VAL_AnInConf_11;
		VALx_AnInFltr_11:= VAL_AnInFltr_11;
		(* <-- Head/TPLC005 AO7*)
		RTU_AnOut_7 := VAL_AnIn_11 / 10;
	end_if;
	if TST_AnIn_12 then
		VALx_AnInConf_12:= VAL_AnInConf_12;
		VALx_AnInFltr_12:= VAL_AnInFltr_12;
		(* <-- Head/TPLC005 AO8*)
		RTU_AnOut_8 := VAL_AnIn_12 / 10;
	end_if;

	if TST_AnOut_1  then
		VALx_AnOut_1 := VAL_AnOut_1;
		VALx_AnOutConf_1 := VAL_AnOutConf_1;
		(* --> Horn2 AI1 + DO4 *)
		VAL2_AnInConf_1 := VAL_AnOutConf_1;
		VAL2_AnInFltr_1 := 16;
		case VAL_AnOutConf_1 of
		1: VAL2_DigOut_4 := 1;
		2: VAL2_DigOut_4 := 0;
		end_case;
	end_if;

	if TST_AnOut_2  then
		VALx_AnOut_2 := VAL_AnOut_2;
		VALx_AnOutConf_2 := VAL_AnOutConf_2;
		(* --> Horn2 AI2 + DO3 *)
		VAL2_AnInConf_2 := VAL_AnOutConf_2;
		VAL2_AnInFltr_2 := 16;
		case VAL_AnOutConf_2 of
		1: VAL2_DigOut_3 := 1;
		2: VAL2_DigOut_3 := 0;
		end_case;
	end_if;

	if TST_AnOut_3  then
		VALx_AnOut_3 := VAL_AnOut_3;
		VALx_AnOutConf_3 := VAL_AnOutConf_3;
		(* --> Head/TPLC005 AI1 *)
		PLC_AnInConf_1 := VAL_AnOutConf_3;
	end_if;

	if TST_AnOut_4  then
		VALx_AnOut_4 := VAL_AnOut_4;
		VALx_AnOutConf_4 := VAL_AnOutConf_4;
		(* --> Head/TPLC005 AI2 *)
		PLC_AnInConf_2 := VAL_AnOutConf_4;
	end_if;

	if TST_Tamb  then
		;
	end_if;

	if TST_RPM  then
		(* <-- Horn2 AO3 PWM *)
		VAL2_AnOutConf_3 := 3; (* PWM *)
		VAL2_AnOut_3 := UINT_TO_INT(VAL_RPM / 10); (* different fixed points *)
	end_if;

	if TST_FWrevision  then
		;
	end_if;

	if TST_HWconfig then
		;
	end_if;

	if TST_RTU1_WR then
		VALx_RTU1_WR := VAL_RTU1_WR;
	end_if;

	if TST_RTU1_RD then
		VAL2_RTUS_WR := VAL_RTU1_RD;
	end_if;

	if TST_RTU3_WR then
		VALx_RTU3_WR := VAL_RTU3_WR;
	end_if;

	if TST_CAN1_WR then
		VALx_CAN1_WR := VAL_CAN1_WR;
	end_if;

	if TST_RTU1_RD then
		;
	end_if;

	if TST_RTU3_RD then
		;
	end_if;

	(* only from the testing equipment *)
	if TST_VCC_set then
		(* --> Head AO3 V *)
		PLC_AnOutConf_3 := 2; (* 0..10 V *)
		PLC_AnOut_3 := VAL_VCC_set; (* FIXME: conversion ? *)
	end_if;

	if TST_mA_max then
		(* --> Head AO4 V *)
		PLC_AnOutConf_4 := 2; (* 0..10 V *)
		PLC_AnOut_4 := VAL_mA_max; (* FIXME: conversion ? *)
	end_if;

	if TST_VCC_fbk then
		(* --> Head AI1 V *)
		PLC_AnInConf_1 := 2; (* 0..10 V *)
	end_if;

	if TST_mA_fbk then
		(* --> Head AI2 V *)
		PLC_AnInConf_2 := 2; (* 0..10 V *)
	end_if;

END_FUNCTION

(* ---- Init.st ---- *)
(*[[
]]*)
PROGRAM Init
#import "Crosstable.gvl"

	PLC_DigDir_8 := False; (* FIXME: empty ? *)
	PLC_DigDir_1 := False; (* PLC_PWR_SWITCH input *)
	PLC_DigDir_2 := True; (* PLC_VPOT_ON output *)
	PLC_DigDir_3 := True; (* PLC_VCC_ON output *)
	PLC_DigDir_4 := False; (* PLC_GO_BUTTON input *)
	RTU_AnOutConf_X := 500; (* ANALOG OUTPUT THRESHOLD *)
	TEST2_COMMAND := TEST_STATUS_LOCAL;
	STATUS := STATUS_IDLE;
	RESULT := RESULT_UNKNOWN;
	if not PLC_DigIn_1 then
		PLC_DigOut_2 := False;
		PLC_DigOut_3 := False;
	end_if;

END_PROGRAM

(* ---- Program1.st ---- *)
(*[[
]]*)
PROGRAM Program1
#import "Crosstable.gvl"
VAR
	first: BOOL;
	(* timer : TON; *)
END_VAR
	if first then
		first := FALSE;

		(* reset all *)
		START2_REMOTE := FALSE;  STARTx_REMOTE := FALSE;
		START2_TEST := FALSE;  STARTx_TEST := FALSE;
		(* POWER ON <-- DO3 *)
		(* OUTPUT ON <-- DO2 *)
		PLC_DigDir_3 := 1;
		PLC_DigDir_2 := 1;
		PLC_DigOut_3 := 0;
		PLC_DigOut_2 := 0;
		(* ANALOG OUTPUT THRESHOLD *)
		RTU_AnOutConf_X := 5;
		STATUS := 0;
	end_if;

	case STATUS of

	0: (* IDLE *)
		if DO_REMOTE then
			START2_REMOTE := TRUE;  STARTx_REMOTE := TRUE;
			STATUS := 1;
		end_if;

	1: (* STARTING *)
		if STATUS2_REMOTE AND STATUSx_REMOTE then
			STATUS := 2;
		end_if;

	2: (* READY *)
		if DO_TEST then
			ClearResults();
			Translate_DigIn();
			Translate_DigOut();
			Translate_AnIn();
			Translate_AnOut();
			Translate_Others();
			(* FIXME: delay? *)
			START2_TEST := TRUE;  STARTx_TEST := TRUE;
			STATUS := 3;
		end_if;
		if not DO_REMOTE then
			START2_REMOTE := FALSE;  STARTx_REMOTE := FALSE;
			STATUS := 6;
		end_if;

	3: (* TESTING *)
		if STATUS2_DONE AND STATUSx_DONE then
			Check_DigIn();
			Check_DigOut();
			Check_AnIn();
			Check_AnOut();
			Check_Others();
			STATUS := 4;
		end_if;

	4: (* DONE *)
		if not DO_TEST then
			START2_TEST := FALSE;  STARTx_TEST := FALSE;
			STATUS := 5;
		end_if;

	5: (* RESETTING *)
		if STATUS2_REMOTE and STATUSx_REMOTE then
			STATUS := 2;
		end_if;

	6: (* STOPPING *)
		if not STATUS2_REMOTE and not STATUSx_REMOTE then
			STATUS := 0;
		end_if;

    else
		(* FIXME: assert *)
		;
    end_case;
END_PROGRAM

(* ---- Testing.st ---- *)
(*[[
]]*)
PROGRAM Testing
#import "Crosstable.gvl"
VAR
	substatus : uint := 0;
	timer : TON;
END_VAR

	case STATUS of

	STATUS_IDLE:
		if (PLC_DigIn_1) then (* PLC_PWR_SWITCH *)
			if (not PLC_DigOut_2) then
				PLC_DigOut_2 := true;
				(* slightly delay the VPOW *)
				return;
			end_if;
			PLC_DigOut_3 := true;
			clearPLC();
			TEST2_COMMAND := TEST_STATUS_REMOTE;
			TEST_STEP := 0;
			RESULT := RESULT_UNKNOWN;
			RESULTS_OK := 0;
			RESULTS_NG := 0;
			STATUS := STATUS_STARTING;
			return;
		end_if;

	STATUS_STARTING:
		if (not PLC_DigIn_1) then
			STATUS := STATUS_STOPPING;
			return;
		end_if;
	    if (TEST2_STATUS = TEST_STATUS_REMOTE and TESTx_STATUS = TEST_STATUS_REMOTE) then
			STATUS := STATUS_READY;
			return;
		end_if;
		timer(IN := TRUE, PT := T#10s); (* boot time *)
		if timer.Q then
			timer(IN := FALSE);
			(* try to rewrite the test starting command *)
		    if (TEST2_STATUS <> TEST_STATUS_REMOTE) then
		        TEST2_COMMAND := TEST_STATUS_REMOTE;
		    end_if;
		    if (TESTx_STATUS <> TEST_STATUS_REMOTE) then
		        TESTx_COMMAND := TEST_STATUS_REMOTE;
		    end_if;
		end_if;

	STATUS_READY:
		(* this state is managed in HMI *)
		substatus := 0;

	STATUS_ERROR:
		(* this state is managed in HMI *)
		;

	STATUS_TESTING:
		if (not PLC_DigIn_1) then
			STATUS := STATUS_STOPPING;
			return;
		end_if;
		case substatus of
		0: (* clear the OK test variables and write the TST ones *)
			ClearOK();
			substatus := 1;
	    1: (* write the TST test variables *)
			WriteTST();
			substatus := 2;
	    2: (* write the VAL test variables *)
			WriteVAL();
			substatus := 3;
	    3: (* wait for propagation of TST and VAL @ priority 3 : 500ms *)
			timer(IN := TRUE, PT := T#500ms);
			if timer.Q then
				timer(IN := FALSE);
				(* write the test starting command *)
		        TEST2_COMMAND := TEST_STATUS_DONE;
		        TESTx_COMMAND := TEST_STATUS_DONE;
				substatus := 4;
			end_if;
	    4: (* wait for propagation of COMMAND @ priority 2 : 500ms and for TPLC005 AnIn *)
			timer(IN := TRUE, PT := T#4500ms); (* 500ms + TPLC005 AnIn slow *)
			if timer.Q then
				timer(IN := FALSE);
				substatus := 5;
			end_if;
		5: (* waiting for test completion and then read the results *)
		    if (TEST2_STATUS = TEST_STATUS_DONE and TESTx_STATUS = TEST_STATUS_DONE) then
				ReadRES();
				substatus := 6; (* need a step for reading RES %Q *)
				return;
			end_if;
		6: (* check RES and VAL *)
			CheckOK();
			substatus := 7;  (* need a step for reading OK %Q *)
		7: (* resume *)
			if AllTestedAreOK() then
				RESULT := RESULT_OK;
				RESULTS_OK := RESULTS_OK + 1;
			else
				RESULT := RESULT_NG;
				RESULTS_NG := RESULTS_NG + 1;
			end_if;
			substatus := 8;
	    8: (* let the hmi visualize the result *)
			timer(IN := TRUE, PT := T#1000ms);
			if timer.Q then
				timer(IN := FALSE);
				STATUS := STATUS_DONE;
			end_if;
		else
			;
		end_case;

	STATUS_DONE:
		if (not PLC_DigIn_1) then
			STATUS := STATUS_STOPPING;
			return;
		end_if;
		if (AUTOMATIC and RESULT = RESULT_OK) or PLC_DigIn_4 then (* GO *)
			ClearPLC();
			STATUS := STATUS_RESETTING;
			return;
		end_if;

	STATUS_RESETTING:
		if (not PLC_DigIn_1) then
			STATUS := STATUS_STOPPING;
			return;
		end_if;
	    if (TEST2_STATUS = TEST_STATUS_REMOTE and TESTx_STATUS = TEST_STATUS_REMOTE) then
			RESULT := RESULT_UNKNOWN;
			STATUS := STATUS_READY;
			return;
		end_if;
		timer(IN := TRUE, PT := T#1s);
		if timer.Q then
			timer(IN := FALSE);
			(* try to rewrite the test resetting command *)
		    if (TEST2_STATUS <> TEST_STATUS_REMOTE) then
		        TEST2_COMMAND := TEST_STATUS_REMOTE;
		    end_if;
		    if (TESTx_STATUS <> TEST_STATUS_REMOTE) then
		        TESTx_COMMAND := TEST_STATUS_REMOTE;
		    end_if;
		end_if;

	STATUS_STOPPING:
		RESULT := RESULT_UNKNOWN;
	    TEST2_COMMAND := TEST_STATUS_LOCAL;
	    TESTx_COMMAND := TEST_STATUS_LOCAL;
		PLC_DigOut_2 := 0;
		PLC_DigOut_3 := 0;
		STATUS := STATUS_IDLE;
		return;

	else
		;
	end_case;

END_PROGRAM
